SPLINE
SPL {X  -146.599, Y  +744.345, Z    +0.000, E1   -36.661, E3 +275980.416}
SPL {X  -158.886, Y  +709.076, Z    +0.000, E1   -22.176, E3 +275984.288}
SPL {X  -161.886, Y  +690.913, Z    +0.000, E1   -12.672, E3 +275988.922}
SPL {X  -162.573, Y  +682.458, Z    +0.000, E1    -7.683, E3 +275988.423}
SPL {X  -162.817, Y  +674.426, Z    +0.000, E1    -2.573, E3 +275988.141}
SPL {X  -162.820, Y  +670.554, Z    +0.000, E1    +0.472, E3 +275987.766}
SPL {X  -162.820, Y  +667.789, Z    +0.000, E1    +3.144, E3 +275987.787}
SPL {X  -162.820, Y  +664.083, Z    +0.000, E1    +7.387, E3 +275987.679}
SPL {X  -162.820, Y  +659.344, Z    +0.000, E1   +13.535, E3 +275987.243}
SPL {X  -162.820, Y  +653.403, Z    +0.000, E1   +21.415, E3 +275987.657}
SPL {X  -162.820, Y  +642.162, Z    +0.000, E1   +35.510, E3 +275986.970}
SPL {X  -162.820, Y  +598.675, Z    +0.000, E1   +56.845, E3 +276004.282}
SPL {X  -162.820, Y  +543.175, Z    +0.000, E1   +54.504, E3 +276080.137}
SPL {X  -162.820, Y  +538.115, Z    +0.000, E1   +53.658, E3 +276093.188}
SPL {X  -162.820, Y  +527.429, Z    +0.000, E1   +53.760, E3 +276108.918}
SPL {X  -162.820, Y  +518.365, Z    +0.000, E1   +53.683, E3 +276123.176}
SPL {X  -162.820, Y  +510.654, Z    +0.000, E1   +53.658, E3 +276135.175}
SPL {X  -162.820, Y  +501.304, Z    +0.000, E1   +53.758, E3 +276148.863}
SPL {X  -162.820, Y  +493.008, Z    +0.000, E1   +53.586, E3 +276162.639}
SPL {X  -162.820, Y  +484.615, Z    +0.000, E1   +53.726, E3 +276174.569}
ENDSPLINE

SPLINE
SPL {X  -162.820, Y  +492.996, Z    +0.000, E1   +49.430, E3 +276187.115}
ENDSPLINE

SPLINE
SPL {X  -162.820, Y  +486.578, Z    +0.000, E1   +49.194, E3 +276199.918}
SPL {X  -162.820, Y  +476.731, Z    +0.000, E1   +50.039, E3 +276212.341}
SPL {X  -162.820, Y  +466.442, Z    +0.000, E1   +50.873, E3 +276225.009}
SPL {X  -162.820, Y  +455.624, Z    +0.000, E1   +51.698, E3 +276238.081}
SPL {X  -162.820, Y  +444.568, Z    +0.000, E1   +52.608, E3 +276250.393}
SPL {X  -162.820, Y  +432.435, Z    +0.000, E1   +53.605, E3 +276263.276}
SPL {X  -162.820, Y  +419.900, Z    +0.000, E1   +54.598, E3 +276275.951}
SPL {X  -162.820, Y  +411.092, Z    +0.000, E1   +54.552, E3 +276289.471}
SPL {X  -162.820, Y  +400.244, Z    +0.000, E1   +54.630, E3 +276304.938}
SPL {X  -162.820, Y  +389.249, Z    +0.000, E1   +54.752, E3 +276320.517}
SPL {X  -162.820, Y  +380.650, Z    +0.000, E1   +54.601, E3 +276333.961}
SPL {X  -162.727, Y  +374.992, Z    +0.000, E1   +54.549, E3 +276342.644}
SPL {X  -162.216, Y  +366.490, Z    +0.000, E1   +54.549, E3 +276355.443}
SPL {X  -161.062, Y  +356.641, Z    +0.000, E1   +54.440, E3 +276370.561}
SPL {X  -159.761, Y  +349.086, Z    +0.000, E1   +54.132, E3 +276383.582}
SPL {X  -158.033, Y  +341.310, Z    +0.000, E1   +53.819, E3 +276396.972}
SPL {X  -156.195, Y  +334.528, Z    +0.000, E1   +53.534, E3 +276408.538}
SPL {X  -154.120, Y  +327.988, Z    +0.000, E1   +53.171, E3 +276420.395}
SPL {X  -151.310, Y  +320.369, Z    +0.000, E1   +52.706, E3 +276434.109}
SPL {X  -148.923, Y  +314.679, Z    +0.000, E1   +52.172, E3 +276445.194}
SPL {X  -146.846, Y  +310.168, Z    +0.000, E1   +51.697, E3 +276454.255}
SPL {X  -140.627, Y  +298.437, Z    +0.000, E1   +54.251, E3 +276458.514}
SPL {X  -122.064, Y  +272.747, Z    +0.000, E1   +48.156, E3 +276564.039}
ENDSPLINE

SPLINE
SPL {X  -148.173, Y  +313.009, Z    +0.000, E1   +35.624, E3 +276647.085}
SPL {X  -158.289, Y  +342.356, Z    +0.000, E1   +23.452, E3 +276650.074}
SPL {X  -161.301, Y  +358.312, Z    +0.000, E1   +15.384, E3 +276652.032}
SPL {X  -162.692, Y  +374.052, Z    +0.000, E1    +6.208, E3 +276651.970}
SPL {X  -162.820, Y  +381.030, Z    +0.000, E1    +1.454, E3 +276652.149}
SPL {X  -162.820, Y  +384.274, Z    +0.000, E1    -1.205, E3 +276651.868}
SPL {X  -162.820, Y  +388.271, Z    +0.000, E1    -5.458, E3 +276651.861}
SPL {X  -162.820, Y  +394.827, Z    +0.000, E1   -13.677, E3 +276651.551}
SPL {X  -162.820, Y  +402.977, Z    +0.000, E1   -24.772, E3 +276651.833}
SPL {X  -162.820, Y  +413.615, Z    +0.000, E1   -37.560, E3 +276651.623}
SPL {X  -162.820, Y  +456.390, Z    +0.000, E1   -57.415, E3 +276668.665}
SPL {X  -162.820, Y  +525.017, Z    +0.000, E1   -58.379, E3 +276739.329}
ENDSPLINE

SPLINE
SPL {X  -162.820, Y  +515.796, Z    +0.000, E1   -54.952, E3 +276748.436}
ENDSPLINE

SPLINE
SPL {X  -162.820, Y  +522.537, Z    +0.000, E1   -55.218, E3 +276756.611}
SPL {X  -162.820, Y  +529.742, Z    +0.000, E1   -55.146, E3 +276767.538}
SPL {X  -162.820, Y  +538.383, Z    +0.000, E1   -55.306, E3 +276778.990}
SPL {X  -162.820, Y  +544.790, Z    +0.000, E1   -55.066, E3 +276789.790}
SPL {X  -162.820, Y  +552.981, Z    +0.000, E1   -55.286, E3 +276800.253}
SPL {X  -162.820, Y  +560.767, Z    +0.000, E1   -55.137, E3 +276812.561}
SPL {X  -162.820, Y  +570.590, Z    +0.000, E1   -55.270, E3 +276825.895}
SPL {X  -162.820, Y  +577.946, Z    +0.000, E1   -55.110, E3 +276837.533}
SPL {X  -162.820, Y  +583.981, Z    +0.000, E1   -55.057, E3 +276846.615}
SPL {X  -162.820, Y  +591.604, Z    +0.000, E1   -55.202, E3 +276856.789}
SPL {X  -162.820, Y  +600.465, Z    +0.000, E1   -55.218, E3 +276869.578}
SPL {X  -162.820, Y  +609.951, Z    +0.000, E1   -55.211, E3 +276883.325}
SPL {X  -162.820, Y  +617.278, Z    +0.000, E1   -55.256, E3 +276893.549}
SPL {X  -162.820, Y  +625.209, Z    +0.000, E1   -55.167, E3 +276905.741}
SPL {X  -162.820, Y  +634.693, Z    +0.000, E1   -55.198, E3 +276919.197}
SPL {X  -162.820, Y  +642.452, Z    +0.000, E1   -55.141, E3 +276930.804}
SPL {X  -162.820, Y  +652.837, Z    +0.000, E1   -55.281, E3 +276945.072}
SPL {X  -162.820, Y  +660.849, Z    +0.000, E1   -55.101, E3 +276957.621}
SPL {X  -162.820, Y  +668.534, Z    +0.000, E1   -55.182, E3 +276968.334}
SPL {X  -162.763, Y  +677.803, Z    +0.000, E1   -55.175, E3 +276981.840}
SPL {X  -162.314, Y  +686.325, Z    +0.000, E1   -55.173, E3 +276994.121}
SPL {X  -161.784, Y  +691.841, Z    +0.000, E1   -55.010, E3 +277003.083}
SPL {X  -161.070, Y  +697.305, Z    +0.000, E1   -54.828, E3 +277012.161}
SPL {X  -159.751, Y  +704.965, Z    +0.000, E1   -54.697, E3 +277024.147}
SPL {X  -158.271, Y  +711.718, Z    +0.000, E1   -54.504, E3 +277034.955}
SPL {X  -157.115, Y  +716.223, Z    +0.000, E1   -54.227, E3 +277043.147}
SPL {X  -154.825, Y  +723.894, Z    +0.000, E1   -53.830, E3 +277056.687}
SPL {X  -152.160, Y  +731.445, Z    +0.000, E1   -53.336, E3 +277070.229}
SPL {X  -149.361, Y  +738.321, Z    +0.000, E1   -52.873, E3 +277082.692}
SPL {X  -146.885, Y  +743.751, Z    +0.000, E1   -52.544, E3 +277092.053}
SPL {X  -144.373, Y  +748.778, Z    +0.000, E1   -52.887, E3 +277097.515}
SPL {X  -137.947, Y  +759.993, Z    +0.000, E1   -55.381, E3 +277100.625}
SPL {X  -123.111, Y  +780.056, Z    +0.000, E1   -48.144, E3 +277199.761}
ENDSPLINE

SPLINE
SPL {X  -146.599, Y  +744.345, Z    +0.000, E1   -36.661, E3 +277284.764}
SPL {X  -157.185, Y  +715.965, Z    +0.000, E1   -25.340, E3 +277287.814}
SPL {X  -159.997, Y  +703.690, Z    +0.000, E1   -19.457, E3 +277289.142}
SPL {X  -161.886, Y  +690.913, Z    +0.000, E1   -12.672, E3 +277293.270}
SPL {X  -162.700, Y  +679.756, Z    +0.000, E1    -6.060, E3 +277292.479}
SPL {X  -162.820, Y  +673.439, Z    +0.000, E1    -1.797, E3 +277292.581}
SPL {X  -162.820, Y  +670.554, Z    +0.000, E1    +0.472, E3 +277292.114}
SPL {X  -162.820, Y  +667.789, Z    +0.000, E1    +3.144, E3 +277292.135}
SPL {X  -162.820, Y  +664.083, Z    +0.000, E1    +7.387, E3 +277292.027}
SPL {X  -162.820, Y  +659.344, Z    +0.000, E1   +13.535, E3 +277291.591}
SPL {X  -162.820, Y  +653.403, Z    +0.000, E1   +21.415, E3 +277292.005}
SPL {X  -162.820, Y  +642.162, Z    +0.000, E1   +35.510, E3 +277291.318}
SPL {X  -162.820, Y  +598.675, Z    +0.000, E1   +56.845, E3 +277308.630}
SPL {X  -162.820, Y  +543.175, Z    +0.000, E1   +54.504, E3 +277384.485}
SPL {X  -162.820, Y  +538.115, Z    +0.000, E1   +53.658, E3 +277397.536}
SPL {X  -162.820, Y  +530.332, Z    +0.000, E1   +53.757, E3 +277408.679}
SPL {X  -162.820, Y  +525.300, Z    +0.000, E1   +53.701, E3 +277416.730}
SPL {X  -162.820, Y  +518.365, Z    +0.000, E1   +53.683, E3 +277427.524}
SPL {X  -162.820, Y  +510.654, Z    +0.000, E1   +53.658, E3 +277439.523}
SPL {X  -162.820, Y  +501.304, Z    +0.000, E1   +53.758, E3 +277453.211}
SPL {X  -162.820, Y  +493.008, Z    +0.000, E1   +53.586, E3 +277466.986}
SPL {X  -162.820, Y  +484.615, Z    +0.000, E1   +53.726, E3 +277478.917}
ENDSPLINE

SPLINE
SPL {X  -162.820, Y  +492.996, Z    +0.000, E1   +49.430, E3 +277491.463}
ENDSPLINE

SPLINE
SPL {X  -162.820, Y  +486.578, Z    +0.000, E1   +49.194, E3 +277504.266}
SPL {X  -162.820, Y  +476.731, Z    +0.000, E1   +50.039, E3 +277516.689}
SPL {X  -162.820, Y  +466.442, Z    +0.000, E1   +50.873, E3 +277529.357}
SPL {X  -162.820, Y  +455.624, Z    +0.000, E1   +51.698, E3 +277542.428}
SPL {X  -162.820, Y  +444.568, Z    +0.000, E1   +52.608, E3 +277554.741}
SPL {X  -162.820, Y  +432.435, Z    +0.000, E1   +53.605, E3 +277567.624}
SPL {X  -162.820, Y  +419.875, Z    +0.000, E1   +54.604, E3 +277580.298}
SPL {X  -162.820, Y  +414.181, Z    +0.000, E1   +54.446, E3 +277589.733}
SPL {X  -162.820, Y  +407.616, Z    +0.000, E1   +54.585, E3 +277598.567}
SPL {X  -162.820, Y  +400.244, Z    +0.000, E1   +54.630, E3 +277609.285}
SPL {X  -162.820, Y  +389.249, Z    +0.000, E1   +54.752, E3 +277624.864}
SPL {X  -162.820, Y  +380.650, Z    +0.000, E1   +54.601, E3 +277638.309}
SPL {X  -162.727, Y  +374.992, Z    +0.000, E1   +54.549, E3 +277646.991}
SPL {X  -162.373, Y  +368.447, Z    +0.000, E1   +54.597, E3 +277656.424}
SPL {X  -161.939, Y  +363.587, Z    +0.000, E1   +54.355, E3 +277665.036}
SPL {X  -160.880, Y  +355.442, Z    +0.000, E1   +54.372, E3 +277677.247}
SPL {X  -159.457, Y  +347.579, Z    +0.000, E1   +54.148, E3 +277689.983}
SPL {X  -158.033, Y  +341.310, Z    +0.000, E1   +53.819, E3 +277701.320}
SPL {X  -156.195, Y  +334.528, Z    +0.000, E1   +53.534, E3 +277712.885}
SPL {X  -154.120, Y  +327.988, Z    +0.000, E1   +53.171, E3 +277724.742}
SPL {X  -151.310, Y  +320.369, Z    +0.000, E1   +52.706, E3 +277738.457}
SPL {X  -148.923, Y  +314.679, Z    +0.000, E1   +52.172, E3 +277749.542}
SPL {X  -146.846, Y  +310.168, Z    +0.000, E1   +51.697, E3 +277758.603}
SPL {X  -140.627, Y  +298.437, Z    +0.000, E1   +54.251, E3 +277762.862}
SPL {X  -122.064, Y  +272.747, Z    +0.000, E1   +48.156, E3 +277868.387}
ENDSPLINE

SPLINE
SPL {X  -148.173, Y  +313.009, Z    +0.000, E1   +35.624, E3 +277951.433}
SPL {X  -159.343, Y  +347.032, Z    +0.000, E1   +21.245, E3 +277955.276}
SPL {X  -161.787, Y  +362.186, Z    +0.000, E1   +13.182, E3 +277956.472}
SPL {X  -162.692, Y  +374.052, Z    +0.000, E1    +6.208, E3 +277956.318}
SPL {X  -162.820, Y  +381.030, Z    +0.000, E1    +1.454, E3 +277956.497}
SPL {X  -162.820, Y  +384.274, Z    +0.000, E1    -1.205, E3 +277956.216}
SPL {X  -162.820, Y  +388.271, Z    +0.000, E1    -5.458, E3 +277956.209}
SPL {X  -162.820, Y  +394.827, Z    +0.000, E1   -13.677, E3 +277955.899}
SPL {X  -162.820, Y  +402.977, Z    +0.000, E1   -24.772, E3 +277956.180}
SPL {X  -162.820, Y  +413.615, Z    +0.000, E1   -37.560, E3 +277955.971}
SPL {X  -162.820, Y  +452.521, Z    +0.000, E1   -56.942, E3 +277970.263}
SPL {X  -162.820, Y  +459.967, Z    +0.000, E1   -57.801, E3 +277975.559}
SPL {X  -162.820, Y  +525.017, Z    +0.000, E1   -58.379, E3 +278043.677}
ENDSPLINE

SPLINE
SPL {X  -162.820, Y  +515.796, Z    +0.000, E1   -54.952, E3 +278052.784}
ENDSPLINE

SPLINE
SPL {X  -162.820, Y  +522.537, Z    +0.000, E1   -55.218, E3 +278060.959}
SPL {X  -162.820, Y  +529.742, Z    +0.000, E1   -55.146, E3 +278071.886}
SPL {X  -162.820, Y  +538.383, Z    +0.000, E1   -55.306, E3 +278083.338}
SPL {X  -162.820, Y  +544.790, Z    +0.000, E1   -55.066, E3 +278094.138}
SPL {X  -162.820, Y  +552.981, Z    +0.000, E1   -55.286, E3 +278104.601}
SPL {X  -162.820, Y  +560.767, Z    +0.000, E1   -55.137, E3 +278116.909}
SPL {X  -162.820, Y  +570.590, Z    +0.000, E1   -55.270, E3 +278130.243}
SPL {X  -162.820, Y  +580.865, Z    +0.000, E1   -55.132, E3 +278146.200}
SPL {X  -162.820, Y  +591.604, Z    +0.000, E1   -55.202, E3 +278161.137}
SPL {X  -162.820, Y  +600.465, Z    +0.000, E1   -55.218, E3 +278173.926}
SPL {X  -162.820, Y  +609.951, Z    +0.000, E1   -55.211, E3 +278187.673}
SPL {X  -162.820, Y  +618.960, Z    +0.000, E1   -55.186, E3 +278200.893}
SPL {X  -162.820, Y  +627.322, Z    +0.000, E1   -55.201, E3 +278212.829}
SPL {X  -162.820, Y  +634.693, Z    +0.000, E1   -55.198, E3 +278223.545}
SPL {X  -162.820, Y  +642.452, Z    +0.000, E1   -55.141, E3 +278235.152}
SPL {X  -162.820, Y  +649.370, Z    +0.000, E1   -55.160, E3 +278245.009}
SPL {X  -162.820, Y  +658.542, Z    +0.000, E1   -55.251, E3 +278257.887}
SPL {X  -162.820, Y  +668.534, Z    +0.000, E1   -55.182, E3 +278272.682}
SPL {X  -162.763, Y  +677.803, Z    +0.000, E1   -55.175, E3 +278286.188}
SPL {X  -162.314, Y  +686.325, Z    +0.000, E1   -55.173, E3 +278298.469}
SPL {X  -161.784, Y  +691.841, Z    +0.000, E1   -55.010, E3 +278307.431}
SPL {X  -161.070, Y  +697.305, Z    +0.000, E1   -54.828, E3 +278316.509}
SPL {X  -159.751, Y  +704.965, Z    +0.000, E1   -54.697, E3 +278328.495}
SPL {X  -158.271, Y  +711.718, Z    +0.000, E1   -54.504, E3 +278339.303}
SPL {X  -157.115, Y  +716.223, Z    +0.000, E1   -54.227, E3 +278347.495}
SPL {X  -155.622, Y  +721.376, Z    +0.000, E1   -53.849, E3 +278357.095}
SPL {X  -153.323, Y  +728.294, Z    +0.000, E1   -53.618, E3 +278368.568}
SPL {X  -150.606, Y  +735.372, Z    +0.000, E1   -53.091, E3 +278381.565}
SPL {X  -148.712, Y  +739.795, Z    +0.000, E1   -52.656, E3 +278390.127}
SPL {X  -146.885, Y  +743.751, Z    +0.000, E1   -52.544, E3 +278396.401}
SPL {X  -144.373, Y  +748.778, Z    +0.000, E1   -52.887, E3 +278401.863}
SPL {X  -137.947, Y  +759.993, Z    +0.000, E1   -55.381, E3 +278404.973}
SPL {X  -123.111, Y  +780.056, Z    +0.000, E1   -48.144, E3 +278504.109}
ENDSPLINE

SPLINE
SPL {X  -146.599, Y  +744.345, Z    +0.000, E1   -36.661, E3 +278589.112}
SPL {X  -158.886, Y  +709.076, Z    +0.000, E1   -22.176, E3 +278592.984}
SPL {X  -161.886, Y  +690.913, Z    +0.000, E1   -12.672, E3 +278597.618}
SPL {X  -162.573, Y  +682.458, Z    +0.000, E1    -7.683, E3 +278597.119}
SPL {X  -162.817, Y  +674.426, Z    +0.000, E1    -2.573, E3 +278596.837}
SPL {X  -162.820, Y  +670.554, Z    +0.000, E1    +0.472, E3 +278596.461}
SPL {X  -162.820, Y  +667.789, Z    +0.000, E1    +3.144, E3 +278596.483}
SPL {X  -162.820, Y  +664.083, Z    +0.000, E1    +7.387, E3 +278596.375}
SPL {X  -162.820, Y  +659.344, Z    +0.000, E1   +13.535, E3 +278595.939}
SPL {X  -162.820, Y  +653.403, Z    +0.000, E1   +21.415, E3 +278596.353}
SPL {X  -162.820, Y  +642.162, Z    +0.000, E1   +35.510, E3 +278595.666}
SPL {X  -162.820, Y  +598.675, Z    +0.000, E1   +56.845, E3 +278612.978}
SPL {X  -162.820, Y  +543.175, Z    +0.000, E1   +54.504, E3 +278688.833}
SPL {X  -162.820, Y  +538.115, Z    +0.000, E1   +53.658, E3 +278701.884}
SPL {X  -162.820, Y  +527.429, Z    +0.000, E1   +53.760, E3 +278717.614}
SPL {X  -162.820, Y  +518.365, Z    +0.000, E1   +53.683, E3 +278731.871}
SPL {X  -162.820, Y  +510.654, Z    +0.000, E1   +53.658, E3 +278743.870}
SPL {X  -162.820, Y  +501.304, Z    +0.000, E1   +53.758, E3 +278757.559}
SPL {X  -162.820, Y  +493.008, Z    +0.000, E1   +53.586, E3 +278771.334}
SPL {X  -162.820, Y  +484.615, Z    +0.000, E1   +53.726, E3 +278783.265}
ENDSPLINE

SPLINE
SPL {X  -162.820, Y  +492.996, Z    +0.000, E1   +49.430, E3 +278795.811}
ENDSPLINE

SPLINE
SPL {X  -162.820, Y  +483.544, Z    +0.000, E1   +49.458, E3 +278812.596}
SPL {X  -162.820, Y  +468.441, Z    +0.000, E1   +50.759, E3 +278831.098}
SPL {X  -162.820, Y  +455.624, Z    +0.000, E1   +51.698, E3 +278846.776}
SPL {X  -162.820, Y  +444.568, Z    +0.000, E1   +52.608, E3 +278859.089}
SPL {X  -162.820, Y  +432.435, Z    +0.000, E1   +53.605, E3 +278871.972}
SPL {X  -162.820, Y  +419.875, Z    +0.000, E1   +54.604, E3 +278884.646}
SPL {X  -162.820, Y  +414.181, Z    +0.000, E1   +54.446, E3 +278894.081}
SPL {X  -162.820, Y  +407.616, Z    +0.000, E1   +54.585, E3 +278902.915}
SPL {X  -162.820, Y  +400.244, Z    +0.000, E1   +54.630, E3 +278913.633}
SPL {X  -162.820, Y  +389.249, Z    +0.000, E1   +54.752, E3 +278929.212}
SPL {X  -162.799, Y  +377.862, Z    +0.000, E1   +54.622, E3 +278946.843}
SPL {X  -162.216, Y  +366.490, Z    +0.000, E1   +54.549, E3 +278964.138}
SPL {X  -160.880, Y  +355.442, Z    +0.000, E1   +54.372, E3 +278981.595}
SPL {X  -159.457, Y  +347.579, Z    +0.000, E1   +54.148, E3 +278994.331}
SPL {X  -158.033, Y  +341.310, Z    +0.000, E1   +53.819, E3 +279005.668}
SPL {X  -155.608, Y  +332.578, Z    +0.000, E1   +53.425, E3 +279020.939}
SPL {X  -152.785, Y  +324.223, Z    +0.000, E1   +52.975, E3 +279035.699}
SPL {X  -150.663, Y  +318.766, Z    +0.000, E1   +52.574, E3 +279045.732}
SPL {X  -148.923, Y  +314.679, Z    +0.000, E1   +52.172, E3 +279053.890}
SPL {X  -146.846, Y  +310.168, Z    +0.000, E1   +51.697, E3 +279062.951}
SPL {X  -140.627, Y  +298.437, Z    +0.000, E1   +54.251, E3 +279067.210}
SPL {X  -122.064, Y  +272.747, Z    +0.000, E1   +48.156, E3 +279172.735}
ENDSPLINE

SPLINE
SPL {X  -148.173, Y  +313.009, Z    +0.000, E1   +35.624, E3 +279255.781}
SPL {X  -158.289, Y  +342.356, Z    +0.000, E1   +23.452, E3 +279258.770}
SPL {X  -161.301, Y  +358.312, Z    +0.000, E1   +15.384, E3 +279260.728}
SPL {X  -162.692, Y  +374.052, Z    +0.000, E1    +6.208, E3 +279260.666}
SPL {X  -162.820, Y  +381.030, Z    +0.000, E1    +1.454, E3 +279260.845}
SPL {X  -162.820, Y  +383.414, Z    +0.000, E1    -0.499, E3 +279260.751}
SPL {X  -162.820, Y  +385.887, Z    +0.000, E1    -2.819, E3 +279260.473}
SPL {X  -162.820, Y  +389.383, Z    +0.000, E1    -6.871, E3 +279260.540}
SPL {X  -162.820, Y  +393.153, Z    +0.000, E1   -11.600, E3 +279260.433}
SPL {X  -162.820, Y  +400.748, Z    +0.000, E1   -21.791, E3 +279260.225}
SPL {X  -162.820, Y  +413.615, Z    +0.000, E1   -37.560, E3 +279260.319}
SPL {X  -162.820, Y  +456.390, Z    +0.000, E1   -57.415, E3 +279277.360}
SPL {X  -162.820, Y  +525.017, Z    +0.000, E1   -58.379, E3 +279348.025}
ENDSPLINE

SPLINE
SPL {X  -162.820, Y  +520.266, Z    +0.000, E1   -55.155, E3 +279362.518}
ENDSPLINE

SPLINE
SPL {X  -162.820, Y  +529.742, Z    +0.000, E1   -55.146, E3 +279376.234}
SPL {X  -162.820, Y  +538.383, Z    +0.000, E1   -55.306, E3 +279387.686}
SPL {X  -162.820, Y  +544.790, Z    +0.000, E1   -55.066, E3 +279398.486}
SPL {X  -162.820, Y  +552.981, Z    +0.000, E1   -55.286, E3 +279408.949}
SPL {X  -162.820, Y  +560.767, Z    +0.000, E1   -55.137, E3 +279421.257}
SPL {X  -162.820, Y  +570.590, Z    +0.000, E1   -55.270, E3 +279434.591}
SPL {X  -162.820, Y  +577.946, Z    +0.000, E1   -55.110, E3 +279446.229}
SPL {X  -162.820, Y  +583.981, Z    +0.000, E1   -55.057, E3 +279455.311}
SPL {X  -162.820, Y  +594.246, Z    +0.000, E1   -55.310, E3 +279468.747}
SPL {X  -162.820, Y  +601.811, Z    +0.000, E1   -55.027, E3 +279481.274}
SPL {X  -162.820, Y  +609.951, Z    +0.000, E1   -55.211, E3 +279492.021}
SPL {X  -162.820, Y  +618.960, Z    +0.000, E1   -55.186, E3 +279505.241}
SPL {X  -162.820, Y  +627.322, Z    +0.000, E1   -55.201, E3 +279517.176}
SPL {X  -162.820, Y  +634.693, Z    +0.000, E1   -55.198, E3 +279527.893}
SPL {X  -162.820, Y  +642.452, Z    +0.000, E1   -55.141, E3 +279539.500}
SPL {X  -162.820, Y  +652.837, Z    +0.000, E1   -55.281, E3 +279553.768}
SPL {X  -162.820, Y  +660.849, Z    +0.000, E1   -55.101, E3 +279566.317}
SPL {X  -162.820, Y  +668.534, Z    +0.000, E1   -55.182, E3 +279577.030}
SPL {X  -162.763, Y  +677.803, Z    +0.000, E1   -55.175, E3 +279590.536}
SPL {X  -162.314, Y  +686.325, Z    +0.000, E1   -55.173, E3 +279602.816}
SPL {X  -161.784, Y  +691.841, Z    +0.000, E1   -55.010, E3 +279611.778}
SPL {X  -161.070, Y  +697.305, Z    +0.000, E1   -54.828, E3 +279620.856}
SPL {X  -159.751, Y  +704.965, Z    +0.000, E1   -54.697, E3 +279632.842}
SPL {X  -158.271, Y  +711.718, Z    +0.000, E1   -54.504, E3 +279643.651}
SPL {X  -157.115, Y  +716.223, Z    +0.000, E1   -54.227, E3 +279651.843}
SPL {X  -155.622, Y  +721.376, Z    +0.000, E1   -53.849, E3 +279661.443}
SPL {X  -153.323, Y  +728.294, Z    +0.000, E1   -53.618, E3 +279672.916}
SPL {X  -150.606, Y  +735.372, Z    +0.000, E1   -53.091, E3 +279685.912}
SPL {X  -148.712, Y  +739.795, Z    +0.000, E1   -52.656, E3 +279694.475}
SPL {X  -146.885, Y  +743.751, Z    +0.000, E1   -52.544, E3 +279700.748}
SPL {X  -144.373, Y  +748.778, Z    +0.000, E1   -52.887, E3 +279706.211}
SPL {X  -137.947, Y  +759.993, Z    +0.000, E1   -55.381, E3 +279709.321}
SPL {X  -123.111, Y  +780.056, Z    +0.000, E1   -48.144, E3 +279808.456}
ENDSPLINE

SPLINE
SPL {X  -146.599, Y  +744.345, Z    +0.000, E1   -36.661, E3 +279893.460}
SPL {X  -158.886, Y  +709.076, Z    +0.000, E1   -22.176, E3 +279897.332}
SPL {X  -161.886, Y  +690.913, Z    +0.000, E1   -12.672, E3 +279901.966}
SPL {X  -162.573, Y  +682.458, Z    +0.000, E1    -7.683, E3 +279901.467}
SPL {X  -162.817, Y  +674.426, Z    +0.000, E1    -2.573, E3 +279901.185}
SPL {X  -162.820, Y  +670.554, Z    +0.000, E1    +0.472, E3 +279900.809}
SPL {X  -162.820, Y  +667.789, Z    +0.000, E1    +3.144, E3 +279900.831}
SPL {X  -162.820, Y  +664.083, Z    +0.000, E1    +7.387, E3 +279900.723}
SPL {X  -162.820, Y  +659.344, Z    +0.000, E1   +13.535, E3 +279900.286}
SPL {X  -162.820, Y  +653.403, Z    +0.000, E1   +21.415, E3 +279900.701}
SPL {X  -162.820, Y  +644.970, Z    +0.000, E1   +32.346, E3 +279900.117}
SPL {X  -162.820, Y  +637.013, Z    +0.000, E1   +41.185, E3 +279899.822}
SPL {X  -162.820, Y  +603.840, Z    +0.000, E1   +55.833, E3 +279914.439}
SPL {X  -162.820, Y  +590.612, Z    +0.000, E1   +58.217, E3 +279921.823}
SPL {X  -162.820, Y  +543.175, Z    +0.000, E1   +54.504, E3 +279993.180}
SPL {X  -162.820, Y  +538.115, Z    +0.000, E1   +53.658, E3 +280006.232}
SPL {X  -162.820, Y  +527.429, Z    +0.000, E1   +53.760, E3 +280021.961}
SPL {X  -162.820, Y  +518.365, Z    +0.000, E1   +53.683, E3 +280036.219}
SPL {X  -162.820, Y  +510.654, Z    +0.000, E1   +53.658, E3 +280048.218}
SPL {X  -162.820, Y  +501.304, Z    +0.000, E1   +53.758, E3 +280061.907}
SPL {X  -162.820, Y  +493.008, Z    +0.000, E1   +53.586, E3 +280075.682}
SPL {X  -162.820, Y  +485.759, Z    +0.000, E1   +53.138, E3 +280089.690}
ENDSPLINE

SPLINE
SPL {X  -162.820, Y  +494.645, Z    +0.000, E1   +48.544, E3 +280102.165}
ENDSPLINE

SPLINE
SPL {X  -162.820, Y  +486.578, Z    +0.000, E1   +49.194, E3 +280112.962}
SPL {X  -162.820, Y  +476.731, Z    +0.000, E1   +50.039, E3 +280125.384}
SPL {X  -162.820, Y  +466.442, Z    +0.000, E1   +50.873, E3 +280138.053}
SPL {X  -162.820, Y  +455.624, Z    +0.000, E1   +51.698, E3 +280151.124}
SPL {X  -162.820, Y  +444.568, Z    +0.000, E1   +52.608, E3 +280163.437}
SPL {X  -162.820, Y  +432.435, Z    +0.000, E1   +53.605, E3 +280176.320}
SPL {X  -162.820, Y  +419.900, Z    +0.000, E1   +54.598, E3 +280188.995}
SPL {X  -162.820, Y  +411.092, Z    +0.000, E1   +54.552, E3 +280202.514}
SPL {X  -162.820, Y  +400.244, Z    +0.000, E1   +54.630, E3 +280217.981}
SPL {X  -162.820, Y  +392.496, Z    +0.000, E1   +54.734, E3 +280228.682}
SPL {X  -162.820, Y  +387.085, Z    +0.000, E1   +54.699, E3 +280236.909}
SPL {X  -162.820, Y  +380.650, Z    +0.000, E1   +54.601, E3 +280247.005}
SPL {X  -162.727, Y  +374.992, Z    +0.000, E1   +54.549, E3 +280255.687}
SPL {X  -162.216, Y  +366.490, Z    +0.000, E1   +54.549, E3 +280268.486}
SPL {X  -160.880, Y  +355.442, Z    +0.000, E1   +54.372, E3 +280285.942}
SPL {X  -159.457, Y  +347.579, Z    +0.000, E1   +54.148, E3 +280298.679}
SPL {X  -158.033, Y  +341.310, Z    +0.000, E1   +53.819, E3 +280310.015}
SPL {X  -155.608, Y  +332.578, Z    +0.000, E1   +53.425, E3 +280325.287}
SPL {X  -153.385, Y  +325.878, Z    +0.000, E1   +53.068, E3 +280336.955}
SPL {X  -151.310, Y  +320.369, Z    +0.000, E1   +52.706, E3 +280347.153}
SPL {X  -148.923, Y  +314.679, Z    +0.000, E1   +52.172, E3 +280358.237}
SPL {X  -146.846, Y  +310.168, Z    +0.000, E1   +51.697, E3 +280367.299}
SPL {X  -140.627, Y  +298.437, Z    +0.000, E1   +54.251, E3 +280371.557}
SPL {X  -122.064, Y  +272.747, Z    +0.000, E1   +48.156, E3 +280477.083}
ENDSPLINE

SPLINE
SPL {X  -148.173, Y  +313.009, Z    +0.000, E1   +35.624, E3 +280560.128}
SPL {X  -158.289, Y  +342.356, Z    +0.000, E1   +23.452, E3 +280563.118}
SPL {X  -161.301, Y  +358.312, Z    +0.000, E1   +15.384, E3 +280565.075}
SPL {X  -162.692, Y  +374.052, Z    +0.000, E1    +6.208, E3 +280565.014}
SPL {X  -162.820, Y  +381.030, Z    +0.000, E1    +1.454, E3 +280565.193}
SPL {X  -162.820, Y  +384.274, Z    +0.000, E1    -1.205, E3 +280564.912}
SPL {X  -162.820, Y  +388.271, Z    +0.000, E1    -5.458, E3 +280564.904}
SPL {X  -162.820, Y  +394.827, Z    +0.000, E1   -13.677, E3 +280564.594}
SPL {X  -162.820, Y  +402.977, Z    +0.000, E1   -24.772, E3 +280564.876}
SPL {X  -162.820, Y  +413.615, Z    +0.000, E1   -37.560, E3 +280564.667}
SPL {X  -162.820, Y  +456.390, Z    +0.000, E1   -57.415, E3 +280581.708}
SPL {X  -162.820, Y  +525.017, Z    +0.000, E1   -58.379, E3 +280652.373}
ENDSPLINE

SPLINE
SPL {X  -162.820, Y  +515.796, Z    +0.000, E1   -54.952, E3 +280661.479}
ENDSPLINE

SPLINE
SPL {X  -162.820, Y  +522.537, Z    +0.000, E1   -55.218, E3 +280669.654}
SPL {X  -162.820, Y  +529.742, Z    +0.000, E1   -55.146, E3 +280680.582}
SPL {X  -162.820, Y  +538.383, Z    +0.000, E1   -55.306, E3 +280692.034}
SPL {X  -162.820, Y  +544.790, Z    +0.000, E1   -55.066, E3 +280702.834}
SPL {X  -162.820, Y  +552.981, Z    +0.000, E1   -55.286, E3 +280713.296}
SPL {X  -162.820, Y  +560.767, Z    +0.000, E1   -55.137, E3 +280725.605}
SPL {X  -162.820, Y  +570.590, Z    +0.000, E1   -55.270, E3 +280738.939}
SPL {X  -162.820, Y  +577.946, Z    +0.000, E1   -55.110, E3 +280750.577}
SPL {X  -162.820, Y  +583.981, Z    +0.000, E1   -55.057, E3 +280759.659}
SPL {X  -162.820, Y  +591.604, Z    +0.000, E1   -55.202, E3 +280769.833}
SPL {X  -162.820, Y  +600.465, Z    +0.000, E1   -55.218, E3 +280782.621}
SPL {X  -162.820, Y  +609.951, Z    +0.000, E1   -55.211, E3 +280796.369}
SPL {X  -162.820, Y  +617.278, Z    +0.000, E1   -55.256, E3 +280806.593}
SPL {X  -162.820, Y  +625.209, Z    +0.000, E1   -55.167, E3 +280818.785}
SPL {X  -162.820, Y  +634.693, Z    +0.000, E1   -55.198, E3 +280832.241}
SPL {X  -162.820, Y  +642.452, Z    +0.000, E1   -55.141, E3 +280843.847}
SPL {X  -162.820, Y  +652.837, Z    +0.000, E1   -55.281, E3 +280858.115}
SPL {X  -162.820, Y  +660.849, Z    +0.000, E1   -55.101, E3 +280870.664}
SPL {X  -162.820, Y  +668.534, Z    +0.000, E1   -55.182, E3 +280881.378}
SPL {X  -162.763, Y  +677.803, Z    +0.000, E1   -55.175, E3 +280894.884}
SPL {X  -162.314, Y  +686.325, Z    +0.000, E1   -55.173, E3 +280907.164}
SPL {X  -161.784, Y  +691.841, Z    +0.000, E1   -55.010, E3 +280916.126}
SPL {X  -161.070, Y  +697.305, Z    +0.000, E1   -54.828, E3 +280925.204}
SPL {X  -159.751, Y  +704.965, Z    +0.000, E1   -54.697, E3 +280937.190}
SPL {X  -158.271, Y  +711.718, Z    +0.000, E1   -54.504, E3 +280947.999}
SPL {X  -157.115, Y  +716.223, Z    +0.000, E1   -54.227, E3 +280956.190}
SPL {X  -154.825, Y  +723.894, Z    +0.000, E1   -53.830, E3 +280969.731}
SPL {X  -152.160, Y  +731.445, Z    +0.000, E1   -53.336, E3 +280983.273}
SPL {X  -149.361, Y  +738.321, Z    +0.000, E1   -52.873, E3 +280995.735}
SPL {X  -146.885, Y  +743.751, Z    +0.000, E1   -52.544, E3 +281005.096}
SPL {X  -144.373, Y  +748.778, Z    +0.000, E1   -52.887, E3 +281010.559}
SPL {X  -137.947, Y  +759.993, Z    +0.000, E1   -55.381, E3 +281013.668}
SPL {X  -123.111, Y  +780.056, Z    +0.000, E1   -48.144, E3 +281112.804}
ENDSPLINE

SPLINE
SPL {X  -146.599, Y  +744.345, Z    +0.000, E1   -36.661, E3 +281197.807}
SPL {X  -157.185, Y  +715.965, Z    +0.000, E1   -25.340, E3 +281200.857}
SPL {X  -159.997, Y  +703.690, Z    +0.000, E1   -19.457, E3 +281202.186}
SPL {X  -161.886, Y  +690.913, Z    +0.000, E1   -12.672, E3 +281206.314}
SPL {X  -162.700, Y  +679.756, Z    +0.000, E1    -6.060, E3 +281205.523}
SPL {X  -162.820, Y  +673.439, Z    +0.000, E1    -1.797, E3 +281205.625}
SPL {X  -162.820, Y  +670.554, Z    +0.000, E1    +0.472, E3 +281205.157}
SPL {X  -162.820, Y  +667.789, Z    +0.000, E1    +3.144, E3 +281205.179}
SPL {X  -162.820, Y  +664.083, Z    +0.000, E1    +7.387, E3 +281205.070}
SPL {X  -162.820, Y  +659.344, Z    +0.000, E1   +13.535, E3 +281204.634}
SPL {X  -162.820, Y  +653.403, Z    +0.000, E1   +21.415, E3 +281205.049}
SPL {X  -162.820, Y  +642.162, Z    +0.000, E1   +35.510, E3 +281204.361}
SPL {X  -162.820, Y  +598.675, Z    +0.000, E1   +56.845, E3 +281221.674}
SPL {X  -162.820, Y  +543.175, Z    +0.000, E1   +54.504, E3 +281297.528}
SPL {X  -162.820, Y  +538.115, Z    +0.000, E1   +53.658, E3 +281310.580}
SPL {X  -162.820, Y  +530.332, Z    +0.000, E1   +53.757, E3 +281321.723}
SPL {X  -162.820, Y  +525.300, Z    +0.000, E1   +53.701, E3 +281329.773}
SPL {X  -162.820, Y  +518.365, Z    +0.000, E1   +53.683, E3 +281340.567}
SPL {X  -162.820, Y  +510.654, Z    +0.000, E1   +53.658, E3 +281352.566}
SPL {X  -162.820, Y  +501.304, Z    +0.000, E1   +53.758, E3 +281366.255}
SPL {X  -162.820, Y  +493.008, Z    +0.000, E1   +53.586, E3 +281380.030}
SPL {X  -162.820, Y  +484.615, Z    +0.000, E1   +53.726, E3 +281391.961}
ENDSPLINE

SPLINE
SPL {X  -162.820, Y  +492.996, Z    +0.000, E1   +49.430, E3 +281404.507}
ENDSPLINE

SPLINE
SPL {X  -162.820, Y  +486.578, Z    +0.000, E1   +49.194, E3 +281417.309}
SPL {X  -162.820, Y  +476.731, Z    +0.000, E1   +50.039, E3 +281429.732}
SPL {X  -162.820, Y  +466.442, Z    +0.000, E1   +50.873, E3 +281442.401}
SPL {X  -162.820, Y  +455.624, Z    +0.000, E1   +51.698, E3 +281455.472}
SPL {X  -162.820, Y  +444.568, Z    +0.000, E1   +52.608, E3 +281467.785}
SPL {X  -162.820, Y  +432.435, Z    +0.000, E1   +53.605, E3 +281480.668}
SPL {X  -162.820, Y  +419.875, Z    +0.000, E1   +54.604, E3 +281493.342}
SPL {X  -162.820, Y  +414.181, Z    +0.000, E1   +54.446, E3 +281502.776}
SPL {X  -162.820, Y  +407.616, Z    +0.000, E1   +54.585, E3 +281511.611}
SPL {X  -162.820, Y  +400.244, Z    +0.000, E1   +54.630, E3 +281522.329}
SPL {X  -162.820, Y  +389.249, Z    +0.000, E1   +54.752, E3 +281537.908}
SPL {X  -162.820, Y  +380.650, Z    +0.000, E1   +54.601, E3 +281551.353}
SPL {X  -162.727, Y  +374.992, Z    +0.000, E1   +54.549, E3 +281560.035}
SPL {X  -162.373, Y  +368.447, Z    +0.000, E1   +54.597, E3 +281569.467}
SPL {X  -161.939, Y  +363.587, Z    +0.000, E1   +54.355, E3 +281578.079}
SPL {X  -161.062, Y  +356.641, Z    +0.000, E1   +54.440, E3 +281587.952}
SPL {X  -159.761, Y  +349.086, Z    +0.000, E1   +54.132, E3 +281600.973}
SPL {X  -158.451, Y  +343.033, Z    +0.000, E1   +53.828, E3 +281611.650}
SPL {X  -156.619, Y  +335.993, Z    +0.000, E1   +53.639, E3 +281623.296}
SPL {X  -154.959, Y  +330.520, Z    +0.000, E1   +53.198, E3 +281633.721}
SPL {X  -153.385, Y  +325.878, Z    +0.000, E1   +53.068, E3 +281641.302}
SPL {X  -151.310, Y  +320.369, Z    +0.000, E1   +52.706, E3 +281651.501}
SPL {X  -148.923, Y  +314.679, Z    +0.000, E1   +52.172, E3 +281662.585}
SPL {X  -146.846, Y  +310.168, Z    +0.000, E1   +51.697, E3 +281671.646}
SPL {X  -140.627, Y  +298.437, Z    +0.000, E1   +54.251, E3 +281675.905}
SPL {X  -122.064, Y  +272.747, Z    +0.000, E1   +48.156, E3 +281781.431}
ENDSPLINE

SPLINE
SPL {X  -148.173, Y  +313.009, Z    +0.000, E1   +35.624, E3 +281864.476}
SPL {X  -159.343, Y  +347.032, Z    +0.000, E1   +21.245, E3 +281868.320}
SPL {X  -162.355, Y  +368.197, Z    +0.000, E1    +9.799, E3 +281869.489}
SPL {X  -162.819, Y  +380.071, Z    +0.000, E1    +2.240, E3 +281869.483}
SPL {X  -162.820, Y  +383.414, Z    +0.000, E1    -0.499, E3 +281869.446}
SPL {X  -162.820, Y  +385.055, Z    +0.000, E1    -2.040, E3 +281869.090}
SPL {X  -162.820, Y  +388.271, Z    +0.000, E1    -5.458, E3 +281869.252}
SPL {X  -162.820, Y  +393.153, Z    +0.000, E1   -11.600, E3 +281869.129}
SPL {X  -162.820, Y  +400.748, Z    +0.000, E1   -21.791, E3 +281868.921}
SPL {X  -162.820, Y  +413.615, Z    +0.000, E1   -37.560, E3 +281869.015}
SPL {X  -162.820, Y  +456.390, Z    +0.000, E1   -57.415, E3 +281886.056}
SPL {X  -162.820, Y  +525.017, Z    +0.000, E1   -58.379, E3 +281956.721}
ENDSPLINE

SPLINE
SPL {X  -162.820, Y  +520.266, Z    +0.000, E1   -55.155, E3 +281971.213}
ENDSPLINE

SPLINE
SPL {X  -162.820, Y  +529.742, Z    +0.000, E1   -55.146, E3 +281984.929}
SPL {X  -162.820, Y  +538.383, Z    +0.000, E1   -55.306, E3 +281996.381}
SPL {X  -162.820, Y  +544.790, Z    +0.000, E1   -55.066, E3 +282007.182}
SPL {X  -162.820, Y  +552.981, Z    +0.000, E1   -55.286, E3 +282017.644}
SPL {X  -162.820, Y  +560.767, Z    +0.000, E1   -55.137, E3 +282029.953}
SPL {X  -162.820, Y  +570.590, Z    +0.000, E1   -55.270, E3 +282043.287}
SPL {X  -162.820, Y  +580.865, Z    +0.000, E1   -55.132, E3 +282059.243}
SPL {X  -162.820, Y  +591.604, Z    +0.000, E1   -55.202, E3 +282074.181}
SPL {X  -162.820, Y  +600.465, Z    +0.000, E1   -55.218, E3 +282086.969}
SPL {X  -162.820, Y  +609.951, Z    +0.000, E1   -55.211, E3 +282100.717}
SPL {X  -162.820, Y  +618.960, Z    +0.000, E1   -55.186, E3 +282113.937}
SPL {X  -162.820, Y  +627.322, Z    +0.000, E1   -55.201, E3 +282125.872}
SPL {X  -162.820, Y  +634.693, Z    +0.000, E1   -55.198, E3 +282136.589}
SPL {X  -162.820, Y  +642.452, Z    +0.000, E1   -55.141, E3 +282148.195}
SPL {X  -162.820, Y  +652.837, Z    +0.000, E1   -55.281, E3 +282162.463}
SPL {X  -162.820, Y  +660.849, Z    +0.000, E1   -55.101, E3 +282175.012}
SPL {X  -162.820, Y  +671.259, Z    +0.000, E1   -55.266, E3 +282189.308}
SPL {X  -162.498, Y  +683.731, Z    +0.000, E1   -55.157, E3 +282208.018}
SPL {X  -161.784, Y  +691.841, Z    +0.000, E1   -55.010, E3 +282220.474}
SPL {X  -161.070, Y  +697.305, Z    +0.000, E1   -54.828, E3 +282229.552}
SPL {X  -159.751, Y  +704.965, Z    +0.000, E1   -54.697, E3 +282241.538}
SPL {X  -158.271, Y  +711.718, Z    +0.000, E1   -54.504, E3 +282252.347}
SPL {X  -157.115, Y  +716.223, Z    +0.000, E1   -54.227, E3 +282260.538}
SPL {X  -155.622, Y  +721.376, Z    +0.000, E1   -53.849, E3 +282270.138}
SPL {X  -153.323, Y  +728.294, Z    +0.000, E1   -53.618, E3 +282281.611}
SPL {X  -150.606, Y  +735.372, Z    +0.000, E1   -53.091, E3 +282294.608}
SPL {X  -148.712, Y  +739.795, Z    +0.000, E1   -52.656, E3 +282303.171}
SPL {X  -146.885, Y  +743.751, Z    +0.000, E1   -52.544, E3 +282309.444}
SPL {X  -144.373, Y  +748.778, Z    +0.000, E1   -52.887, E3 +282314.907}
SPL {X  -137.947, Y  +759.993, Z    +0.000, E1   -55.381, E3 +282318.016}
SPL {X  -123.111, Y  +780.056, Z    +0.000, E1   -48.144, E3 +282417.152}
ENDSPLINE

SPLINE
SPL {X  -146.599, Y  +744.345, Z    +0.000, E1   -36.661, E3 +282502.155}
SPL {X  -157.185, Y  +715.965, Z    +0.000, E1   -25.340, E3 +282505.205}
SPL {X  -159.997, Y  +703.690, Z    +0.000, E1   -19.457, E3 +282506.533}
SPL {X  -161.886, Y  +690.913, Z    +0.000, E1   -12.672, E3 +282510.661}
SPL {X  -162.700, Y  +679.756, Z    +0.000, E1    -6.060, E3 +282509.871}
SPL {X  -162.820, Y  +673.439, Z    +0.000, E1    -1.797, E3 +282509.973}
SPL {X  -162.820, Y  +670.554, Z    +0.000, E1    +0.472, E3 +282509.505}
SPL {X  -162.820, Y  +667.789, Z    +0.000, E1    +3.144, E3 +282509.527}
SPL {X  -162.820, Y  +664.083, Z    +0.000, E1    +7.387, E3 +282509.418}
SPL {X  -162.820, Y  +659.344, Z    +0.000, E1   +13.535, E3 +282508.982}
SPL {X  -162.820, Y  +653.403, Z    +0.000, E1   +21.415, E3 +282509.397}
SPL {X  -162.820, Y  +642.162, Z    +0.000, E1   +35.510, E3 +282508.709}
SPL {X  -162.820, Y  +598.675, Z    +0.000, E1   +56.845, E3 +282526.022}
SPL {X  -162.820, Y  +543.175, Z    +0.000, E1   +54.504, E3 +282601.876}
SPL {X  -162.820, Y  +538.115, Z    +0.000, E1   +53.658, E3 +282614.927}
SPL {X  -162.820, Y  +527.429, Z    +0.000, E1   +53.760, E3 +282630.657}
SPL {X  -162.820, Y  +518.365, Z    +0.000, E1   +53.683, E3 +282644.915}
SPL {X  -162.820, Y  +508.465, Z    +0.000, E1   +53.706, E3 +282660.129}
SPL {X  -162.820, Y  +499.206, Z    +0.000, E1   +53.779, E3 +282673.569}
SPL {X  -162.820, Y  +493.008, Z    +0.000, E1   +53.586, E3 +282684.378}
SPL {X  -162.820, Y  +485.759, Z    +0.000, E1   +53.138, E3 +282698.385}
ENDSPLINE

SPLINE
SPL {X  -162.820, Y  +494.645, Z    +0.000, E1   +48.544, E3 +282710.861}
ENDSPLINE

SPLINE
SPL {X  -162.820, Y  +486.578, Z    +0.000, E1   +49.194, E3 +282721.657}
SPL {X  -162.820, Y  +476.731, Z    +0.000, E1   +50.039, E3 +282734.080}
SPL {X  -162.820, Y  +466.442, Z    +0.000, E1   +50.873, E3 +282746.749}
SPL {X  -162.820, Y  +455.624, Z    +0.000, E1   +51.698, E3 +282759.820}
SPL {X  -162.820, Y  +444.568, Z    +0.000, E1   +52.608, E3 +282772.133}
SPL {X  -162.820, Y  +432.435, Z    +0.000, E1   +53.605, E3 +282785.016}
SPL {X  -162.820, Y  +419.875, Z    +0.000, E1   +54.604, E3 +282797.690}
SPL {X  -162.820, Y  +414.181, Z    +0.000, E1   +54.446, E3 +282807.124}
SPL {X  -162.820, Y  +407.616, Z    +0.000, E1   +54.585, E3 +282815.958}
SPL {X  -162.820, Y  +400.244, Z    +0.000, E1   +54.630, E3 +282826.677}
SPL {X  -162.820, Y  +389.249, Z    +0.000, E1   +54.752, E3 +282842.256}
SPL {X  -162.799, Y  +377.862, Z    +0.000, E1   +54.622, E3 +282859.886}
SPL {X  -162.216, Y  +366.490, Z    +0.000, E1   +54.549, E3 +282877.182}
SPL {X  -160.880, Y  +355.442, Z    +0.000, E1   +54.372, E3 +282894.638}
SPL {X  -159.457, Y  +347.579, Z    +0.000, E1   +54.148, E3 +282907.375}
SPL {X  -158.033, Y  +341.310, Z    +0.000, E1   +53.819, E3 +282918.711}
SPL {X  -155.608, Y  +332.578, Z    +0.000, E1   +53.425, E3 +282933.983}
SPL {X  -152.785, Y  +324.223, Z    +0.000, E1   +52.975, E3 +282948.742}
SPL {X  -150.663, Y  +318.766, Z    +0.000, E1   +52.574, E3 +282958.775}
SPL {X  -148.923, Y  +314.679, Z    +0.000, E1   +52.172, E3 +282966.933}
SPL {X  -146.846, Y  +310.168, Z    +0.000, E1   +51.697, E3 +282975.994}
SPL {X  -140.627, Y  +298.437, Z    +0.000, E1   +54.251, E3 +282980.253}
SPL {X  -122.064, Y  +272.747, Z    +0.000, E1   +48.156, E3 +283085.779}
ENDSPLINE

SPLINE
SPL {X  -148.173, Y  +313.009, Z    +0.000, E1   +35.624, E3 +283168.824}
SPL {X  -158.289, Y  +342.356, Z    +0.000, E1   +23.452, E3 +283171.814}
SPL {X  -161.301, Y  +358.312, Z    +0.000, E1   +15.384, E3 +283173.771}
SPL {X  -162.692, Y  +374.052, Z    +0.000, E1    +6.208, E3 +283173.709}
SPL {X  -162.820, Y  +381.030, Z    +0.000, E1    +1.454, E3 +283173.888}
SPL {X  -162.820, Y  +384.274, Z    +0.000, E1    -1.205, E3 +283173.607}
SPL {X  -162.820, Y  +388.271, Z    +0.000, E1    -5.458, E3 +283173.600}
SPL {X  -162.820, Y  +394.827, Z    +0.000, E1   -13.677, E3 +283173.290}
SPL {X  -162.820, Y  +402.977, Z    +0.000, E1   -24.772, E3 +283173.572}
SPL {X  -162.820, Y  +413.615, Z    +0.000, E1   -37.560, E3 +283173.362}
SPL {X  -162.820, Y  +456.390, Z    +0.000, E1   -57.415, E3 +283190.404}
SPL {X  -162.820, Y  +525.017, Z    +0.000, E1   -58.379, E3 +283261.069}
ENDSPLINE

SPLINE
SPL {X  -162.820, Y  +515.796, Z    +0.000, E1   -54.952, E3 +283270.175}
ENDSPLINE

SPLINE
SPL {X  -162.820, Y  +522.537, Z    +0.000, E1   -55.218, E3 +283278.350}
SPL {X  -162.820, Y  +529.742, Z    +0.000, E1   -55.146, E3 +283289.277}
SPL {X  -162.820, Y  +538.383, Z    +0.000, E1   -55.306, E3 +283300.729}
SPL {X  -162.820, Y  +544.790, Z    +0.000, E1   -55.066, E3 +283311.530}
SPL {X  -162.820, Y  +552.981, Z    +0.000, E1   -55.286, E3 +283321.992}
SPL {X  -162.820, Y  +560.767, Z    +0.000, E1   -55.137, E3 +283334.300}
SPL {X  -162.820, Y  +570.590, Z    +0.000, E1   -55.270, E3 +283347.634}
SPL {X  -162.820, Y  +577.946, Z    +0.000, E1   -55.110, E3 +283359.272}
SPL {X  -162.820, Y  +583.981, Z    +0.000, E1   -55.057, E3 +283368.355}
SPL {X  -162.820, Y  +594.246, Z    +0.000, E1   -55.310, E3 +283381.790}
SPL {X  -162.820, Y  +601.811, Z    +0.000, E1   -55.027, E3 +283394.318}
SPL {X  -162.820, Y  +609.951, Z    +0.000, E1   -55.211, E3 +283405.064}
SPL {X  -162.820, Y  +617.278, Z    +0.000, E1   -55.256, E3 +283415.289}
SPL {X  -162.820, Y  +625.209, Z    +0.000, E1   -55.167, E3 +283427.480}
SPL {X  -162.820, Y  +634.693, Z    +0.000, E1   -55.198, E3 +283440.937}
SPL {X  -162.820, Y  +642.452, Z    +0.000, E1   -55.141, E3 +283452.543}
SPL {X  -162.820, Y  +652.837, Z    +0.000, E1   -55.281, E3 +283466.811}
SPL {X  -162.820, Y  +660.849, Z    +0.000, E1   -55.101, E3 +283479.360}
SPL {X  -162.820, Y  +668.534, Z    +0.000, E1   -55.182, E3 +283490.074}
SPL {X  -162.763, Y  +677.803, Z    +0.000, E1   -55.175, E3 +283503.580}
SPL {X  -162.314, Y  +686.325, Z    +0.000, E1   -55.173, E3 +283515.860}
SPL {X  -161.784, Y  +691.841, Z    +0.000, E1   -55.010, E3 +283524.822}
SPL {X  -160.705, Y  +699.660, Z    +0.000, E1   -54.830, E3 +283537.482}
SPL {X  -158.809, Y  +709.418, Z    +0.000, E1   -54.602, E3 +283552.954}
SPL {X  -157.115, Y  +716.223, Z    +0.000, E1   -54.227, E3 +283564.886}
SPL {X  -154.825, Y  +723.894, Z    +0.000, E1   -53.830, E3 +283578.426}
SPL {X  -152.160, Y  +731.445, Z    +0.000, E1   -53.336, E3 +283591.968}
SPL {X  -150.059, Y  +736.687, Z    +0.000, E1   -53.023, E3 +283601.134}
SPL {X  -147.746, Y  +741.922, Z    +0.000, E1   -52.631, E3 +283610.842}
SPL {X  -144.373, Y  +748.778, Z    +0.000, E1   -52.887, E3 +283619.255}
SPL {X  -137.947, Y  +759.993, Z    +0.000, E1   -55.381, E3 +283622.364}
SPL {X  -123.111, Y  +780.056, Z    +0.000, E1   -48.144, E3 +283721.500}
ENDSPLINE

SPLINE
SPL {X  -146.599, Y  +744.345, Z    +0.000, E1   -36.661, E3 +283806.503}
SPL {X  -158.886, Y  +709.076, Z    +0.000, E1   -22.176, E3 +283810.375}
SPL {X  -161.886, Y  +690.913, Z    +0.000, E1   -12.672, E3 +283815.009}
SPL {X  -162.573, Y  +682.458, Z    +0.000, E1    -7.683, E3 +283814.510}
SPL {X  -162.817, Y  +674.426, Z    +0.000, E1    -2.573, E3 +283814.228}
SPL {X  -162.820, Y  +670.554, Z    +0.000, E1    +0.472, E3 +283813.853}
SPL {X  -162.820, Y  +667.789, Z    +0.000, E1    +3.144, E3 +283813.874}
SPL {X  -162.820, Y  +664.083, Z    +0.000, E1    +7.387, E3 +283813.766}
SPL {X  -162.820, Y  +659.344, Z    +0.000, E1   +13.535, E3 +283813.330}
SPL {X  -162.820, Y  +653.403, Z    +0.000, E1   +21.415, E3 +283813.744}
SPL {X  -162.820, Y  +642.162, Z    +0.000, E1   +35.510, E3 +283813.057}
SPL {X  -162.820, Y  +598.675, Z    +0.000, E1   +56.845, E3 +283830.369}
SPL {X  -162.820, Y  +543.175, Z    +0.000, E1   +54.504, E3 +283906.224}
SPL {X  -162.820, Y  +538.115, Z    +0.000, E1   +53.658, E3 +283919.275}
SPL {X  -162.820, Y  +527.429, Z    +0.000, E1   +53.760, E3 +283935.005}
SPL {X  -162.820, Y  +518.365, Z    +0.000, E1   +53.683, E3 +283949.263}
SPL {X  -162.820, Y  +510.654, Z    +0.000, E1   +53.658, E3 +283961.262}
SPL {X  -162.820, Y  +501.304, Z    +0.000, E1   +53.758, E3 +283974.950}
SPL {X  -162.820, Y  +493.008, Z    +0.000, E1   +53.586, E3 +283988.726}
SPL {X  -162.820, Y  +485.759, Z    +0.000, E1   +53.138, E3 +284002.733}
ENDSPLINE

SPLINE
SPL {X  -162.820, Y  +494.645, Z    +0.000, E1   +48.544, E3 +284015.209}
ENDSPLINE

SPLINE
SPL {X  -162.820, Y  +483.544, Z    +0.000, E1   +49.458, E3 +284029.987}
SPL {X  -162.820, Y  +468.441, Z    +0.000, E1   +50.759, E3 +284048.489}
SPL {X  -162.820, Y  +455.624, Z    +0.000, E1   +51.698, E3 +284064.167}
SPL {X  -162.820, Y  +444.568, Z    +0.000, E1   +52.608, E3 +284076.480}
SPL {X  -162.820, Y  +432.435, Z    +0.000, E1   +53.605, E3 +284089.363}
SPL {X  -162.820, Y  +419.900, Z    +0.000, E1   +54.598, E3 +284102.038}
SPL {X  -162.820, Y  +411.092, Z    +0.000, E1   +54.552, E3 +284115.558}
SPL {X  -162.820, Y  +400.244, Z    +0.000, E1   +54.630, E3 +284131.025}
SPL {X  -162.820, Y  +389.249, Z    +0.000, E1   +54.752, E3 +284146.604}
SPL {X  -162.820, Y  +380.650, Z    +0.000, E1   +54.601, E3 +284160.048}
SPL {X  -162.727, Y  +374.992, Z    +0.000, E1   +54.549, E3 +284168.730}
SPL {X  -162.216, Y  +366.490, Z    +0.000, E1   +54.549, E3 +284181.530}
SPL {X  -161.062, Y  +356.641, Z    +0.000, E1   +54.440, E3 +284196.648}
SPL {X  -159.761, Y  +349.086, Z    +0.000, E1   +54.132, E3 +284209.669}
SPL {X  -158.033, Y  +341.310, Z    +0.000, E1   +53.819, E3 +284223.059}
SPL {X  -155.608, Y  +332.578, Z    +0.000, E1   +53.425, E3 +284238.330}
SPL {X  -153.385, Y  +325.878, Z    +0.000, E1   +53.068, E3 +284249.998}
SPL {X  -151.310, Y  +320.369, Z    +0.000, E1   +52.706, E3 +284260.196}
SPL {X  -148.923, Y  +314.679, Z    +0.000, E1   +52.172, E3 +284271.281}
SPL {X  -146.846, Y  +310.168, Z    +0.000, E1   +51.697, E3 +284280.342}
SPL {X  -140.627, Y  +298.437, Z    +0.000, E1   +54.251, E3 +284284.601}
SPL {X  -122.064, Y  +272.747, Z    +0.000, E1   +48.156, E3 +284390.126}
ENDSPLINE

SPLINE
SPL {X  -148.173, Y  +313.009, Z    +0.000, E1   +35.624, E3 +284473.172}
SPL {X  -159.343, Y  +347.032, Z    +0.000, E1   +21.245, E3 +284477.015}
SPL {X  -161.787, Y  +362.186, Z    +0.000, E1   +13.182, E3 +284478.211}
SPL {X  -162.692, Y  +374.052, Z    +0.000, E1    +6.208, E3 +284478.057}
SPL {X  -162.820, Y  +382.143, Z    +0.000, E1    +0.693, E3 +284478.192}
SPL {X  -162.820, Y  +385.055, Z    +0.000, E1    -2.040, E3 +284477.786}
SPL {X  -162.820, Y  +388.271, Z    +0.000, E1    -5.458, E3 +284477.948}
SPL {X  -162.820, Y  +393.153, Z    +0.000, E1   -11.600, E3 +284477.825}
SPL {X  -162.820, Y  +400.748, Z    +0.000, E1   -21.791, E3 +284477.616}
SPL {X  -162.820, Y  +413.615, Z    +0.000, E1   -37.560, E3 +284477.710}
SPL {X  -162.820, Y  +452.521, Z    +0.000, E1   -56.942, E3 +284492.002}
SPL {X  -162.820, Y  +459.967, Z    +0.000, E1   -57.801, E3 +284497.298}
SPL {X  -162.820, Y  +525.017, Z    +0.000, E1   -58.379, E3 +284565.416}
ENDSPLINE

SPLINE
SPL {X  -162.820, Y  +520.266, Z    +0.000, E1   -55.155, E3 +284579.909}
ENDSPLINE

SPLINE
SPL {X  -162.820, Y  +529.742, Z    +0.000, E1   -55.146, E3 +284593.625}
SPL {X  -162.820, Y  +538.383, Z    +0.000, E1   -55.306, E3 +284605.077}
SPL {X  -162.820, Y  +544.790, Z    +0.000, E1   -55.066, E3 +284615.877}
SPL {X  -162.820, Y  +555.105, Z    +0.000, E1   -55.222, E3 +284629.998}
SPL {X  -162.820, Y  +563.355, Z    +0.000, E1   -55.172, E3 +284642.064}
SPL {X  -162.820, Y  +570.590, Z    +0.000, E1   -55.270, E3 +284651.982}
SPL {X  -162.820, Y  +580.865, Z    +0.000, E1   -55.132, E3 +284667.939}
SPL {X  -162.820, Y  +594.246, Z    +0.000, E1   -55.310, E3 +284686.138}
SPL {X  -162.820, Y  +601.811, Z    +0.000, E1   -55.027, E3 +284698.666}
SPL {X  -162.820, Y  +609.951, Z    +0.000, E1   -55.211, E3 +284709.412}
SPL {X  -162.820, Y  +618.960, Z    +0.000, E1   -55.186, E3 +284722.632}
SPL {X  -162.820, Y  +627.322, Z    +0.000, E1   -55.201, E3 +284734.568}
SPL {X  -162.820, Y  +634.693, Z    +0.000, E1   -55.198, E3 +284745.284}
SPL {X  -162.820, Y  +642.452, Z    +0.000, E1   -55.141, E3 +284756.891}
SPL {X  -162.820, Y  +649.370, Z    +0.000, E1   -55.160, E3 +284766.748}
SPL {X  -162.820, Y  +658.542, Z    +0.000, E1   -55.251, E3 +284779.626}
SPL {X  -162.820, Y  +671.259, Z    +0.000, E1   -55.266, E3 +284798.003}
SPL {X  -162.498, Y  +683.731, Z    +0.000, E1   -55.157, E3 +284816.713}
SPL {X  -161.784, Y  +691.841, Z    +0.000, E1   -55.010, E3 +284829.170}
SPL {X  -161.070, Y  +697.305, Z    +0.000, E1   -54.828, E3 +284838.248}
SPL {X  -159.751, Y  +704.965, Z    +0.000, E1   -54.697, E3 +284850.234}
SPL {X  -158.271, Y  +711.718, Z    +0.000, E1   -54.504, E3 +284861.042}
SPL {X  -157.115, Y  +716.223, Z    +0.000, E1   -54.227, E3 +284869.234}
SPL {X  -154.825, Y  +723.894, Z    +0.000, E1   -53.830, E3 +284882.774}
SPL {X  -152.160, Y  +731.445, Z    +0.000, E1   -53.336, E3 +284896.316}
SPL {X  -150.059, Y  +736.687, Z    +0.000, E1   -53.023, E3 +284905.482}
SPL {X  -147.746, Y  +741.922, Z    +0.000, E1   -52.631, E3 +284915.189}
SPL {X  -144.373, Y  +748.778, Z    +0.000, E1   -52.887, E3 +284923.602}
SPL {X  -137.947, Y  +759.993, Z    +0.000, E1   -55.381, E3 +284926.712}
SPL {X  -123.111, Y  +780.056, Z    +0.000, E1   -48.144, E3 +285025.848}
ENDSPLINE

SPLINE
SPL {X  -146.599, Y  +744.345, Z    +0.000, E1   -36.661, E3 +285110.851}
SPL {X  -157.185, Y  +715.965, Z    +0.000, E1   -25.340, E3 +285113.901}
SPL {X  -159.997, Y  +703.690, Z    +0.000, E1   -19.457, E3 +285115.229}
SPL {X  -161.886, Y  +690.913, Z    +0.000, E1   -12.672, E3 +285119.357}
SPL {X  -162.700, Y  +679.756, Z    +0.000, E1    -6.060, E3 +285118.566}
SPL {X  -162.820, Y  +673.439, Z    +0.000, E1    -1.797, E3 +285118.668}
SPL {X  -162.820, Y  +670.554, Z    +0.000, E1    +0.472, E3 +285118.201}
SPL {X  -162.820, Y  +667.789, Z    +0.000, E1    +3.144, E3 +285118.222}
SPL {X  -162.820, Y  +664.083, Z    +0.000, E1    +7.387, E3 +285118.114}
SPL {X  -162.820, Y  +659.344, Z    +0.000, E1   +13.535, E3 +285117.678}
SPL {X  -162.820, Y  +653.403, Z    +0.000, E1   +21.415, E3 +285118.092}
SPL {X  -162.820, Y  +642.162, Z    +0.000, E1   +35.510, E3 +285117.405}
SPL {X  -162.820, Y  +598.675, Z    +0.000, E1   +56.845, E3 +285134.717}
SPL {X  -162.820, Y  +542.287, Z    +0.000, E1   +54.257, E3 +285213.621}
SPL {X  -162.820, Y  +533.839, Z    +0.000, E1   +53.682, E3 +285230.042}
SPL {X  -162.820, Y  +525.300, Z    +0.000, E1   +53.701, E3 +285242.817}
SPL {X  -162.820, Y  +518.365, Z    +0.000, E1   +53.683, E3 +285253.611}
SPL {X  -162.820, Y  +510.654, Z    +0.000, E1   +53.658, E3 +285265.610}
SPL {X  -162.820, Y  +501.304, Z    +0.000, E1   +53.758, E3 +285279.298}
SPL {X  -162.820, Y  +493.008, Z    +0.000, E1   +53.586, E3 +285293.073}
SPL {X  -162.820, Y  +485.759, Z    +0.000, E1   +53.138, E3 +285307.081}
ENDSPLINE

SPLINE
SPL {X  -162.820, Y  +494.645, Z    +0.000, E1   +48.544, E3 +285319.557}
ENDSPLINE

SPLINE
SPL {X  -162.820, Y  +486.578, Z    +0.000, E1   +49.194, E3 +285330.353}
SPL {X  -162.820, Y  +476.731, Z    +0.000, E1   +50.039, E3 +285342.776}
SPL {X  -162.820, Y  +466.442, Z    +0.000, E1   +50.873, E3 +285355.444}
SPL {X  -162.820, Y  +455.624, Z    +0.000, E1   +51.698, E3 +285368.515}
SPL {X  -162.820, Y  +444.568, Z    +0.000, E1   +52.608, E3 +285380.828}
SPL {X  -162.820, Y  +432.435, Z    +0.000, E1   +53.605, E3 +285393.711}
SPL {X  -162.820, Y  +419.900, Z    +0.000, E1   +54.598, E3 +285406.386}
SPL {X  -162.820, Y  +411.092, Z    +0.000, E1   +54.552, E3 +285419.906}
SPL {X  -162.820, Y  +400.244, Z    +0.000, E1   +54.630, E3 +285435.372}
SPL {X  -162.820, Y  +389.249, Z    +0.000, E1   +54.752, E3 +285450.951}
SPL {X  -162.799, Y  +377.862, Z    +0.000, E1   +54.622, E3 +285468.582}
SPL {X  -162.373, Y  +368.447, Z    +0.000, E1   +54.597, E3 +285482.511}
SPL {X  -161.939, Y  +363.587, Z    +0.000, E1   +54.355, E3 +285491.123}
SPL {X  -161.062, Y  +356.641, Z    +0.000, E1   +54.440, E3 +285500.996}
SPL {X  -159.761, Y  +349.086, Z    +0.000, E1   +54.132, E3 +285514.017}
SPL {X  -158.451, Y  +343.033, Z    +0.000, E1   +53.828, E3 +285524.693}
SPL {X  -156.619, Y  +335.993, Z    +0.000, E1   +53.639, E3 +285536.340}
SPL {X  -154.959, Y  +330.520, Z    +0.000, E1   +53.198, E3 +285546.765}
SPL {X  -153.385, Y  +325.878, Z    +0.000, E1   +53.068, E3 +285554.346}
SPL {X  -151.310, Y  +320.369, Z    +0.000, E1   +52.706, E3 +285564.544}
SPL {X  -148.923, Y  +314.679, Z    +0.000, E1   +52.172, E3 +285575.629}
SPL {X  -146.846, Y  +310.168, Z    +0.000, E1   +51.697, E3 +285584.690}
SPL {X  -140.627, Y  +298.437, Z    +0.000, E1   +54.251, E3 +285588.949}
SPL {X  -122.064, Y  +272.747, Z    +0.000, E1   +48.156, E3 +285694.474}
ENDSPLINE

SPLINE
SPL {X  -148.173, Y  +313.009, Z    +0.000, E1   +35.624, E3 +285777.520}
SPL {X  -159.343, Y  +347.032, Z    +0.000, E1   +21.245, E3 +285781.363}
SPL {X  -162.355, Y  +368.197, Z    +0.000, E1    +9.799, E3 +285782.532}
SPL {X  -162.819, Y  +380.071, Z    +0.000, E1    +2.240, E3 +285782.527}
SPL {X  -162.820, Y  +383.414, Z    +0.000, E1    -0.499, E3 +285782.490}
SPL {X  -162.820, Y  +385.887, Z    +0.000, E1    -2.819, E3 +285782.212}
SPL {X  -162.820, Y  +389.383, Z    +0.000, E1    -6.871, E3 +285782.279}
SPL {X  -162.820, Y  +393.153, Z    +0.000, E1   -11.600, E3 +285782.172}
SPL {X  -162.820, Y  +400.748, Z    +0.000, E1   -21.791, E3 +285781.964}
SPL {X  -162.820, Y  +413.615, Z    +0.000, E1   -37.560, E3 +285782.058}
SPL {X  -162.820, Y  +456.390, Z    +0.000, E1   -57.415, E3 +285799.099}
SPL {X  -162.820, Y  +525.017, Z    +0.000, E1   -58.379, E3 +285869.764}
ENDSPLINE

SPLINE
SPL {X  -162.820, Y  +520.266, Z    +0.000, E1   -55.155, E3 +285884.257}
ENDSPLINE

SPLINE
SPL {X  -162.820, Y  +529.742, Z    +0.000, E1   -55.146, E3 +285897.973}
SPL {X  -162.820, Y  +538.383, Z    +0.000, E1   -55.306, E3 +285909.425}
SPL {X  -162.820, Y  +544.790, Z    +0.000, E1   -55.066, E3 +285920.225}
SPL {X  -162.820, Y  +552.981, Z    +0.000, E1   -55.286, E3 +285930.688}
SPL {X  -162.820, Y  +560.767, Z    +0.000, E1   -55.137, E3 +285942.996}
SPL {X  -162.820, Y  +570.590, Z    +0.000, E1   -55.270, E3 +285956.330}
SPL {X  -162.820, Y  +577.946, Z    +0.000, E1   -55.110, E3 +285967.968}
SPL {X  -162.820, Y  +583.981, Z    +0.000, E1   -55.057, E3 +285977.050}
SPL {X  -162.820, Y  +594.246, Z    +0.000, E1   -55.310, E3 +285990.486}
SPL {X  -162.820, Y  +601.811, Z    +0.000, E1   -55.027, E3 +286003.014}
SPL {X  -162.820, Y  +609.951, Z    +0.000, E1   -55.211, E3 +286013.760}
SPL {X  -162.820, Y  +618.960, Z    +0.000, E1   -55.186, E3 +286026.980}
SPL {X  -162.820, Y  +627.322, Z    +0.000, E1   -55.201, E3 +286038.916}
SPL {X  -162.820, Y  +634.693, Z    +0.000, E1   -55.198, E3 +286049.632}
SPL {X  -162.820, Y  +642.452, Z    +0.000, E1   -55.141, E3 +286061.239}
SPL {X  -162.820, Y  +652.837, Z    +0.000, E1   -55.281, E3 +286075.507}
SPL {X  -162.820, Y  +660.849, Z    +0.000, E1   -55.101, E3 +286088.056}
SPL {X  -162.820, Y  +668.534, Z    +0.000, E1   -55.182, E3 +286098.769}
SPL {X  -162.763, Y  +677.803, Z    +0.000, E1   -55.175, E3 +286112.275}
SPL {X  -162.084, Y  +688.960, Z    +0.000, E1   -55.150, E3 +286128.730}
SPL {X  -161.070, Y  +697.305, Z    +0.000, E1   -54.828, E3 +286142.595}
SPL {X  -159.751, Y  +704.965, Z    +0.000, E1   -54.697, E3 +286154.582}
SPL {X  -158.271, Y  +711.718, Z    +0.000, E1   -54.504, E3 +286165.390}
SPL {X  -157.115, Y  +716.223, Z    +0.000, E1   -54.227, E3 +286173.582}
SPL {X  -155.622, Y  +721.376, Z    +0.000, E1   -53.849, E3 +286183.182}
SPL {X  -153.323, Y  +728.294, Z    +0.000, E1   -53.618, E3 +286194.655}
SPL {X  -150.606, Y  +735.372, Z    +0.000, E1   -53.091, E3 +286207.652}
SPL {X  -148.712, Y  +739.795, Z    +0.000, E1   -52.656, E3 +286216.214}
SPL {X  -146.885, Y  +743.751, Z    +0.000, E1   -52.544, E3 +286222.488}
SPL {X  -144.373, Y  +748.778, Z    +0.000, E1   -52.887, E3 +286227.950}
SPL {X  -137.947, Y  +759.993, Z    +0.000, E1   -55.381, E3 +286231.060}
SPL {X  -123.111, Y  +780.056, Z    +0.000, E1   -48.144, E3 +286330.195}
ENDSPLINE

SPLINE
SPL {X  -146.599, Y  +744.345, Z    +0.000, E1   -36.661, E3 +286415.199}
SPL {X  -158.886, Y  +709.076, Z    +0.000, E1   -22.176, E3 +286419.071}
SPL {X  -161.886, Y  +690.913, Z    +0.000, E1   -12.672, E3 +286423.705}
SPL {X  -162.573, Y  +682.458, Z    +0.000, E1    -7.683, E3 +286423.206}
SPL {X  -162.817, Y  +674.426, Z    +0.000, E1    -2.573, E3 +286422.924}
SPL {X  -162.820, Y  +670.554, Z    +0.000, E1    +0.472, E3 +286422.548}
SPL {X  -162.820, Y  +667.789, Z    +0.000, E1    +3.144, E3 +286422.570}
SPL {X  -162.820, Y  +664.083, Z    +0.000, E1    +7.387, E3 +286422.462}
SPL {X  -162.820, Y  +659.344, Z    +0.000, E1   +13.535, E3 +286422.025}
SPL {X  -162.820, Y  +653.403, Z    +0.000, E1   +21.415, E3 +286422.440}
SPL {X  -162.820, Y  +642.162, Z    +0.000, E1   +35.510, E3 +286421.753}
SPL {X  -162.820, Y  +598.675, Z    +0.000, E1   +56.845, E3 +286439.065}
SPL {X  -162.820, Y  +543.175, Z    +0.000, E1   +54.504, E3 +286514.919}
SPL {X  -162.820, Y  +538.115, Z    +0.000, E1   +53.658, E3 +286527.971}
SPL {X  -162.820, Y  +527.429, Z    +0.000, E1   +53.760, E3 +286543.701}
SPL {X  -162.820, Y  +518.365, Z    +0.000, E1   +53.683, E3 +286557.958}
SPL {X  -162.820, Y  +510.654, Z    +0.000, E1   +53.658, E3 +286569.957}
SPL {X  -162.820, Y  +501.304, Z    +0.000, E1   +53.758, E3 +286583.646}
SPL {X  -162.820, Y  +493.008, Z    +0.000, E1   +53.586, E3 +286597.421}
SPL {X  -162.820, Y  +484.615, Z    +0.000, E1   +53.726, E3 +286609.352}
ENDSPLINE

SPLINE
SPL {X  -162.820, Y  +492.996, Z    +0.000, E1   +49.430, E3 +286621.898}
ENDSPLINE

SPLINE
SPL {X  -162.820, Y  +486.578, Z    +0.000, E1   +49.194, E3 +286634.701}
SPL {X  -162.820, Y  +476.731, Z    +0.000, E1   +50.039, E3 +286647.124}
SPL {X  -162.820, Y  +466.442, Z    +0.000, E1   +50.873, E3 +286659.792}
SPL {X  -162.820, Y  +455.624, Z    +0.000, E1   +51.698, E3 +286672.863}
SPL {X  -162.820, Y  +444.568, Z    +0.000, E1   +52.608, E3 +286685.176}
SPL {X  -162.820, Y  +432.435, Z    +0.000, E1   +53.605, E3 +286698.059}
SPL {X  -162.820, Y  +419.900, Z    +0.000, E1   +54.598, E3 +286710.734}
SPL {X  -162.820, Y  +411.092, Z    +0.000, E1   +54.552, E3 +286724.254}
SPL {X  -162.820, Y  +400.244, Z    +0.000, E1   +54.630, E3 +286739.720}
SPL {X  -162.820, Y  +389.249, Z    +0.000, E1   +54.752, E3 +286755.299}
SPL {X  -162.820, Y  +380.650, Z    +0.000, E1   +54.601, E3 +286768.744}
SPL {X  -162.727, Y  +374.992, Z    +0.000, E1   +54.549, E3 +286777.426}
SPL {X  -162.216, Y  +366.490, Z    +0.000, E1   +54.549, E3 +286790.225}
SPL {X  -161.062, Y  +356.641, Z    +0.000, E1   +54.440, E3 +286805.343}
SPL {X  -159.761, Y  +349.086, Z    +0.000, E1   +54.132, E3 +286818.365}
SPL {X  -158.033, Y  +341.310, Z    +0.000, E1   +53.819, E3 +286831.755}
SPL {X  -156.195, Y  +334.528, Z    +0.000, E1   +53.534, E3 +286843.320}
SPL {X  -154.120, Y  +327.988, Z    +0.000, E1   +53.171, E3 +286855.177}
SPL {X  -151.310, Y  +320.369, Z    +0.000, E1   +52.706, E3 +286868.892}
SPL {X  -148.923, Y  +314.679, Z    +0.000, E1   +52.172, E3 +286879.977}
SPL {X  -146.846, Y  +310.168, Z    +0.000, E1   +51.697, E3 +286889.038}
SPL {X  -140.627, Y  +298.437, Z    +0.000, E1   +54.251, E3 +286893.297}
SPL {X  -122.064, Y  +272.747, Z    +0.000, E1   +48.156, E3 +286998.822}
ENDSPLINE

SPLINE
SPL {X  -148.173, Y  +313.009, Z    +0.000, E1   +35.624, E3 +287081.867}
SPL {X  -158.289, Y  +342.356, Z    +0.000, E1   +23.452, E3 +287084.857}
SPL {X  -161.301, Y  +358.312, Z    +0.000, E1   +15.384, E3 +287086.815}
SPL {X  -162.692, Y  +374.052, Z    +0.000, E1    +6.208, E3 +287086.753}
SPL {X  -162.820, Y  +381.030, Z    +0.000, E1    +1.454, E3 +287086.932}
SPL {X  -162.820, Y  +384.274, Z    +0.000, E1    -1.205, E3 +287086.651}
SPL {X  -162.820, Y  +388.271, Z    +0.000, E1    -5.458, E3 +287086.643}
SPL {X  -162.820, Y  +394.827, Z    +0.000, E1   -13.677, E3 +287086.333}
SPL {X  -162.820, Y  +402.977, Z    +0.000, E1   -24.772, E3 +287086.615}
SPL {X  -162.820, Y  +413.615, Z    +0.000, E1   -37.560, E3 +287086.406}
SPL {X  -162.820, Y  +456.390, Z    +0.000, E1   -57.415, E3 +287103.447}
SPL {X  -162.820, Y  +525.017, Z    +0.000, E1   -58.379, E3 +287174.112}
ENDSPLINE

SPLINE
SPL {X  -162.820, Y  +515.796, Z    +0.000, E1   -54.952, E3 +287183.219}
ENDSPLINE

SPLINE
SPL {X  -162.820, Y  +522.537, Z    +0.000, E1   -55.218, E3 +287191.394}
SPL {X  -162.820, Y  +529.742, Z    +0.000, E1   -55.146, E3 +287202.321}
SPL {X  -162.820, Y  +538.383, Z    +0.000, E1   -55.306, E3 +287213.773}
SPL {X  -162.820, Y  +544.790, Z    +0.000, E1   -55.066, E3 +287224.573}
SPL {X  -162.820, Y  +552.981, Z    +0.000, E1   -55.286, E3 +287235.035}
SPL {X  -162.820, Y  +560.767, Z    +0.000, E1   -55.137, E3 +287247.344}
SPL {X  -162.820, Y  +570.590, Z    +0.000, E1   -55.270, E3 +287260.678}
SPL {X  -162.820, Y  +577.946, Z    +0.000, E1   -55.110, E3 +287272.316}
SPL {X  -162.820, Y  +583.981, Z    +0.000, E1   -55.057, E3 +287281.398}
SPL {X  -162.820, Y  +591.604, Z    +0.000, E1   -55.202, E3 +287291.572}
SPL {X  -162.820, Y  +600.465, Z    +0.000, E1   -55.218, E3 +287304.360}
SPL {X  -162.820, Y  +609.951, Z    +0.000, E1   -55.211, E3 +287318.108}
SPL {X  -162.820, Y  +617.278, Z    +0.000, E1   -55.256, E3 +287328.332}
SPL {X  -162.820, Y  +625.209, Z    +0.000, E1   -55.167, E3 +287340.524}
SPL {X  -162.820, Y  +634.693, Z    +0.000, E1   -55.198, E3 +287353.980}
SPL {X  -162.820, Y  +642.452, Z    +0.000, E1   -55.141, E3 +287365.587}
SPL {X  -162.820, Y  +652.837, Z    +0.000, E1   -55.281, E3 +287379.855}
SPL {X  -162.820, Y  +660.849, Z    +0.000, E1   -55.101, E3 +287392.403}
SPL {X  -162.820, Y  +668.534, Z    +0.000, E1   -55.182, E3 +287403.117}
SPL {X  -162.763, Y  +677.803, Z    +0.000, E1   -55.175, E3 +287416.623}
SPL {X  -162.314, Y  +686.325, Z    +0.000, E1   -55.173, E3 +287428.903}
SPL {X  -161.784, Y  +691.841, Z    +0.000, E1   -55.010, E3 +287437.865}
SPL {X  -161.070, Y  +697.305, Z    +0.000, E1   -54.828, E3 +287446.943}
SPL {X  -159.751, Y  +704.965, Z    +0.000, E1   -54.697, E3 +287458.929}
SPL {X  -158.271, Y  +711.718, Z    +0.000, E1   -54.504, E3 +287469.738}
SPL {X  -157.115, Y  +716.223, Z    +0.000, E1   -54.227, E3 +287477.930}
SPL {X  -155.622, Y  +721.376, Z    +0.000, E1   -53.849, E3 +287487.530}
SPL {X  -153.323, Y  +728.294, Z    +0.000, E1   -53.618, E3 +287499.003}
SPL {X  -150.606, Y  +735.372, Z    +0.000, E1   -53.091, E3 +287511.999}
SPL {X  -148.712, Y  +739.795, Z    +0.000, E1   -52.656, E3 +287520.562}
SPL {X  -146.885, Y  +743.751, Z    +0.000, E1   -52.544, E3 +287526.835}
SPL {X  -144.373, Y  +748.778, Z    +0.000, E1   -52.887, E3 +287532.298}
SPL {X  -137.947, Y  +759.993, Z    +0.000, E1   -55.381, E3 +287535.408}
SPL {X  -123.111, Y  +780.056, Z    +0.000, E1   -48.144, E3 +287634.543}
ENDSPLINE

SPLINE
SPL {X  -146.599, Y  +744.345, Z    +0.000, E1   -36.661, E3 +287719.547}
SPL {X  -158.886, Y  +709.076, Z    +0.000, E1   -22.176, E3 +287723.419}
SPL {X  -161.886, Y  +690.913, Z    +0.000, E1   -12.672, E3 +287728.053}
SPL {X  -162.573, Y  +682.458, Z    +0.000, E1    -7.683, E3 +287727.554}
SPL {X  -162.817, Y  +674.426, Z    +0.000, E1    -2.573, E3 +287727.272}
SPL {X  -162.820, Y  +670.554, Z    +0.000, E1    +0.472, E3 +287726.896}
SPL {X  -162.820, Y  +667.789, Z    +0.000, E1    +3.144, E3 +287726.918}
SPL {X  -162.820, Y  +664.083, Z    +0.000, E1    +7.387, E3 +287726.810}
SPL {X  -162.820, Y  +659.344, Z    +0.000, E1   +13.535, E3 +287726.373}
SPL {X  -162.820, Y  +653.403, Z    +0.000, E1   +21.415, E3 +287726.788}
SPL {X  -162.820, Y  +642.162, Z    +0.000, E1   +35.510, E3 +287726.100}
SPL {X  -162.820, Y  +598.675, Z    +0.000, E1   +56.845, E3 +287743.413}
SPL {X  -162.820, Y  +543.175, Z    +0.000, E1   +54.504, E3 +287819.267}
SPL {X  -162.820, Y  +538.115, Z    +0.000, E1   +53.658, E3 +287832.319}
SPL {X  -162.820, Y  +527.429, Z    +0.000, E1   +53.760, E3 +287848.048}
SPL {X  -162.820, Y  +518.365, Z    +0.000, E1   +53.683, E3 +287862.306}
SPL {X  -162.820, Y  +510.654, Z    +0.000, E1   +53.658, E3 +287874.305}
SPL {X  -162.820, Y  +501.304, Z    +0.000, E1   +53.758, E3 +287887.994}
SPL {X  -162.820, Y  +493.008, Z    +0.000, E1   +53.586, E3 +287901.769}
SPL {X  -162.820, Y  +484.615, Z    +0.000, E1   +53.726, E3 +287913.700}
ENDSPLINE

SPLINE
SPL {X  -162.820, Y  +492.996, Z    +0.000, E1   +49.430, E3 +287926.246}
ENDSPLINE

SPLINE
SPL {X  -162.820, Y  +483.544, Z    +0.000, E1   +49.458, E3 +287943.030}
SPL {X  -162.820, Y  +468.441, Z    +0.000, E1   +50.759, E3 +287961.533}
SPL {X  -162.820, Y  +455.624, Z    +0.000, E1   +51.698, E3 +287977.211}
SPL {X  -162.820, Y  +444.568, Z    +0.000, E1   +52.608, E3 +287989.524}
SPL {X  -162.820, Y  +432.435, Z    +0.000, E1   +53.605, E3 +288002.407}
SPL {X  -162.820, Y  +419.900, Z    +0.000, E1   +54.598, E3 +288015.081}
SPL {X  -162.820, Y  +411.092, Z    +0.000, E1   +54.552, E3 +288028.601}
SPL {X  -162.820, Y  +400.244, Z    +0.000, E1   +54.630, E3 +288044.068}
SPL {X  -162.820, Y  +389.249, Z    +0.000, E1   +54.752, E3 +288059.647}
SPL {X  -162.820, Y  +380.650, Z    +0.000, E1   +54.601, E3 +288073.092}
SPL {X  -162.727, Y  +374.992, Z    +0.000, E1   +54.549, E3 +288081.774}
SPL {X  -162.373, Y  +368.447, Z    +0.000, E1   +54.597, E3 +288091.206}
SPL {X  -161.939, Y  +363.587, Z    +0.000, E1   +54.355, E3 +288099.818}
SPL {X  -161.062, Y  +356.641, Z    +0.000, E1   +54.440, E3 +288109.691}
SPL {X  -159.761, Y  +349.086, Z    +0.000, E1   +54.132, E3 +288122.712}
SPL {X  -158.033, Y  +341.310, Z    +0.000, E1   +53.819, E3 +288136.102}
SPL {X  -156.195, Y  +334.528, Z    +0.000, E1   +53.534, E3 +288147.668}
SPL {X  -154.120, Y  +327.988, Z    +0.000, E1   +53.171, E3 +288159.525}
SPL {X  -151.310, Y  +320.369, Z    +0.000, E1   +52.706, E3 +288173.240}
SPL {X  -148.923, Y  +314.679, Z    +0.000, E1   +52.172, E3 +288184.324}
SPL {X  -146.846, Y  +310.168, Z    +0.000, E1   +51.697, E3 +288193.386}
SPL {X  -140.627, Y  +298.437, Z    +0.000, E1   +54.251, E3 +288197.644}
SPL {X  -122.064, Y  +272.747, Z    +0.000, E1   +48.156, E3 +288303.170}
ENDSPLINE

SPLINE
SPL {X  -148.173, Y  +313.009, Z    +0.000, E1   +35.624, E3 +288386.215}
SPL {X  -159.343, Y  +347.032, Z    +0.000, E1   +21.245, E3 +288390.059}
SPL {X  -162.355, Y  +368.197, Z    +0.000, E1    +9.799, E3 +288391.228}
SPL {X  -162.819, Y  +380.071, Z    +0.000, E1    +2.240, E3 +288391.222}
SPL {X  -162.820, Y  +383.414, Z    +0.000, E1    -0.499, E3 +288391.185}
SPL {X  -162.820, Y  +385.887, Z    +0.000, E1    -2.819, E3 +288390.908}
SPL {X  -162.820, Y  +389.383, Z    +0.000, E1    -6.871, E3 +288390.975}
SPL {X  -162.820, Y  +393.153, Z    +0.000, E1   -11.600, E3 +288390.868}
SPL {X  -162.820, Y  +400.748, Z    +0.000, E1   -21.791, E3 +288390.660}
SPL {X  -162.820, Y  +413.615, Z    +0.000, E1   -37.560, E3 +288390.754}
SPL {X  -162.820, Y  +456.390, Z    +0.000, E1   -57.415, E3 +288407.795}
SPL {X  -162.820, Y  +525.017, Z    +0.000, E1   -58.379, E3 +288478.460}
ENDSPLINE

SPLINE
SPL {X  -162.820, Y  +520.266, Z    +0.000, E1   -55.155, E3 +288492.952}
ENDSPLINE

SPLINE
SPL {X  -162.820, Y  +529.742, Z    +0.000, E1   -55.146, E3 +288506.669}
SPL {X  -162.820, Y  +538.383, Z    +0.000, E1   -55.306, E3 +288518.121}
SPL {X  -162.820, Y  +544.790, Z    +0.000, E1   -55.066, E3 +288528.921}
SPL {X  -162.820, Y  +552.981, Z    +0.000, E1   -55.286, E3 +288539.383}
SPL {X  -162.820, Y  +560.767, Z    +0.000, E1   -55.137, E3 +288551.692}
SPL {X  -162.820, Y  +570.590, Z    +0.000, E1   -55.270, E3 +288565.026}
SPL {X  -162.820, Y  +577.946, Z    +0.000, E1   -55.110, E3 +288576.663}
SPL {X  -162.820, Y  +583.981, Z    +0.000, E1   -55.057, E3 +288585.746}
SPL {X  -162.820, Y  +594.246, Z    +0.000, E1   -55.310, E3 +288599.181}
SPL {X  -162.820, Y  +601.811, Z    +0.000, E1   -55.027, E3 +288611.709}
SPL {X  -162.820, Y  +609.951, Z    +0.000, E1   -55.211, E3 +288622.456}
SPL {X  -162.820, Y  +618.960, Z    +0.000, E1   -55.186, E3 +288635.676}
SPL {X  -162.820, Y  +627.322, Z    +0.000, E1   -55.201, E3 +288647.611}
SPL {X  -162.820, Y  +634.693, Z    +0.000, E1   -55.198, E3 +288658.328}
SPL {X  -162.820, Y  +642.452, Z    +0.000, E1   -55.141, E3 +288669.934}
SPL {X  -162.820, Y  +652.837, Z    +0.000, E1   -55.281, E3 +288684.202}
SPL {X  -162.820, Y  +660.849, Z    +0.000, E1   -55.101, E3 +288696.751}
SPL {X  -162.820, Y  +668.534, Z    +0.000, E1   -55.182, E3 +288707.465}
SPL {X  -162.763, Y  +677.803, Z    +0.000, E1   -55.175, E3 +288720.971}
SPL {X  -162.084, Y  +688.960, Z    +0.000, E1   -55.150, E3 +288737.426}
SPL {X  -161.070, Y  +697.305, Z    +0.000, E1   -54.828, E3 +288751.291}
SPL {X  -159.751, Y  +704.965, Z    +0.000, E1   -54.697, E3 +288763.277}
SPL {X  -158.271, Y  +711.718, Z    +0.000, E1   -54.504, E3 +288774.086}
SPL {X  -157.115, Y  +716.223, Z    +0.000, E1   -54.227, E3 +288782.277}
SPL {X  -155.622, Y  +721.376, Z    +0.000, E1   -53.849, E3 +288791.877}
SPL {X  -154.043, Y  +726.236, Z    +0.000, E1   -53.722, E3 +288799.626}
SPL {X  -152.160, Y  +731.445, Z    +0.000, E1   -53.336, E3 +288809.360}
SPL {X  -149.361, Y  +738.321, Z    +0.000, E1   -52.873, E3 +288821.822}
SPL {X  -145.628, Y  +746.320, Z    +0.000, E1   -52.740, E3 +288833.940}
SPL {X  -137.947, Y  +759.993, Z    +0.000, E1   -55.381, E3 +288839.755}
SPL {X  -123.111, Y  +780.056, Z    +0.000, E1   -48.144, E3 +288938.891}
ENDSPLINE

SPLINE
SPL {X  -146.599, Y  +744.345, Z    +0.000, E1   -36.661, E3 +289023.894}
SPL {X  -157.185, Y  +715.965, Z    +0.000, E1   -25.340, E3 +289026.944}
SPL {X  -159.997, Y  +703.690, Z    +0.000, E1   -19.457, E3 +289028.273}
SPL {X  -161.886, Y  +690.913, Z    +0.000, E1   -12.672, E3 +289032.401}
SPL {X  -162.700, Y  +679.756, Z    +0.000, E1    -6.060, E3 +289031.610}
SPL {X  -162.820, Y  +673.439, Z    +0.000, E1    -1.797, E3 +289031.712}
SPL {X  -162.820, Y  +670.554, Z    +0.000, E1    +0.472, E3 +289031.244}
SPL {X  -162.820, Y  +667.789, Z    +0.000, E1    +3.144, E3 +289031.266}
SPL {X  -162.820, Y  +664.083, Z    +0.000, E1    +7.387, E3 +289031.157}
SPL {X  -162.820, Y  +659.344, Z    +0.000, E1   +13.535, E3 +289030.721}
SPL {X  -162.820, Y  +653.403, Z    +0.000, E1   +21.415, E3 +289031.136}
SPL {X  -162.820, Y  +642.162, Z    +0.000, E1   +35.510, E3 +289030.448}
SPL {X  -162.820, Y  +598.675, Z    +0.000, E1   +56.845, E3 +289047.761}
SPL {X  -162.820, Y  +542.287, Z    +0.000, E1   +54.257, E3 +289126.664}
SPL {X  -162.820, Y  +533.839, Z    +0.000, E1   +53.682, E3 +289143.085}
SPL {X  -162.820, Y  +525.300, Z    +0.000, E1   +53.701, E3 +289155.860}
SPL {X  -162.820, Y  +518.365, Z    +0.000, E1   +53.683, E3 +289166.654}
SPL {X  -162.820, Y  +510.654, Z    +0.000, E1   +53.658, E3 +289178.653}
SPL {X  -162.820, Y  +501.304, Z    +0.000, E1   +53.758, E3 +289192.342}
SPL {X  -162.820, Y  +493.008, Z    +0.000, E1   +53.586, E3 +289206.117}
SPL {X  -162.820, Y  +485.759, Z    +0.000, E1   +53.138, E3 +289220.124}
ENDSPLINE

SPLINE
SPL {X  -162.820, Y  +494.645, Z    +0.000, E1   +48.544, E3 +289232.600}
ENDSPLINE

SPLINE
SPL {X  -162.820, Y  +486.578, Z    +0.000, E1   +49.194, E3 +289243.396}
SPL {X  -162.820, Y  +476.731, Z    +0.000, E1   +50.039, E3 +289255.819}
SPL {X  -162.820, Y  +466.442, Z    +0.000, E1   +50.873, E3 +289268.488}
SPL {X  -162.820, Y  +455.624, Z    +0.000, E1   +51.698, E3 +289281.559}
SPL {X  -162.820, Y  +444.568, Z    +0.000, E1   +52.608, E3 +289293.872}
SPL {X  -162.820, Y  +432.435, Z    +0.000, E1   +53.605, E3 +289306.755}
SPL {X  -162.820, Y  +419.875, Z    +0.000, E1   +54.604, E3 +289319.429}
SPL {X  -162.820, Y  +414.181, Z    +0.000, E1   +54.446, E3 +289328.863}
SPL {X  -162.820, Y  +407.616, Z    +0.000, E1   +54.585, E3 +289337.697}
SPL {X  -162.820, Y  +400.244, Z    +0.000, E1   +54.630, E3 +289348.416}
SPL {X  -162.820, Y  +389.249, Z    +0.000, E1   +54.752, E3 +289363.995}
SPL {X  -162.799, Y  +377.862, Z    +0.000, E1   +54.622, E3 +289381.625}
SPL {X  -162.373, Y  +368.447, Z    +0.000, E1   +54.597, E3 +289395.554}
SPL {X  -161.939, Y  +363.587, Z    +0.000, E1   +54.355, E3 +289404.166}
SPL {X  -161.062, Y  +356.641, Z    +0.000, E1   +54.440, E3 +289414.039}
SPL {X  -159.761, Y  +349.086, Z    +0.000, E1   +54.132, E3 +289427.060}
SPL {X  -158.451, Y  +343.033, Z    +0.000, E1   +53.828, E3 +289437.737}
SPL {X  -156.619, Y  +335.993, Z    +0.000, E1   +53.639, E3 +289449.383}
SPL {X  -154.959, Y  +330.520, Z    +0.000, E1   +53.198, E3 +289459.808}
SPL {X  -152.785, Y  +324.223, Z    +0.000, E1   +52.975, E3 +289470.481}
SPL {X  -150.663, Y  +318.766, Z    +0.000, E1   +52.574, E3 +289480.514}
SPL {X  -148.923, Y  +314.679, Z    +0.000, E1   +52.172, E3 +289488.672}
SPL {X  -146.846, Y  +310.168, Z    +0.000, E1   +51.697, E3 +289497.733}
SPL {X  -140.627, Y  +298.437, Z    +0.000, E1   +54.251, E3 +289501.992}
SPL {X  -122.064, Y  +272.747, Z    +0.000, E1   +48.156, E3 +289607.518}
ENDSPLINE

SPLINE
SPL {X  -143.204, Y  +303.021, Z    +0.000, E1   +38.944, E3 +289687.814}
SPL {X  -149.792, Y  +316.682, Z    +0.000, E1   +34.282, E3 +289691.392}
SPL {X  -159.343, Y  +347.032, Z    +0.000, E1   +21.245, E3 +289694.407}
SPL {X  -162.355, Y  +368.197, Z    +0.000, E1    +9.799, E3 +289695.576}
SPL {X  -162.819, Y  +380.071, Z    +0.000, E1    +2.240, E3 +289695.570}
SPL {X  -162.820, Y  +383.414, Z    +0.000, E1    -0.499, E3 +289695.533}
SPL {X  -162.820, Y  +385.055, Z    +0.000, E1    -2.040, E3 +289695.177}
SPL {X  -162.820, Y  +388.271, Z    +0.000, E1    -5.458, E3 +289695.339}
SPL {X  -162.820, Y  +394.827, Z    +0.000, E1   -13.677, E3 +289695.029}
SPL {X  -162.820, Y  +402.977, Z    +0.000, E1   -24.772, E3 +289695.311}
SPL {X  -162.820, Y  +413.615, Z    +0.000, E1   -37.560, E3 +289695.102}
SPL {X  -162.820, Y  +456.390, Z    +0.000, E1   -57.415, E3 +289712.143}
SPL {X  -162.820, Y  +525.017, Z    +0.000, E1   -58.379, E3 +289782.808}
ENDSPLINE

SPLINE
SPL {X  -162.820, Y  +515.796, Z    +0.000, E1   -54.952, E3 +289791.914}
ENDSPLINE

SPLINE
SPL {X  -162.820, Y  +522.537, Z    +0.000, E1   -55.218, E3 +289800.089}
SPL {X  -162.820, Y  +529.742, Z    +0.000, E1   -55.146, E3 +289811.016}
SPL {X  -162.820, Y  +538.383, Z    +0.000, E1   -55.306, E3 +289822.468}
SPL {X  -162.820, Y  +544.790, Z    +0.000, E1   -55.066, E3 +289833.269}
SPL {X  -162.820, Y  +552.981, Z    +0.000, E1   -55.286, E3 +289843.731}
SPL {X  -162.820, Y  +560.767, Z    +0.000, E1   -55.137, E3 +289856.040}
SPL {X  -162.820, Y  +570.590, Z    +0.000, E1   -55.270, E3 +289869.374}
SPL {X  -162.820, Y  +577.946, Z    +0.000, E1   -55.110, E3 +289881.011}
SPL {X  -162.820, Y  +583.981, Z    +0.000, E1   -55.057, E3 +289890.094}
SPL {X  -162.820, Y  +591.604, Z    +0.000, E1   -55.202, E3 +289900.268}
SPL {X  -162.820, Y  +600.465, Z    +0.000, E1   -55.218, E3 +289913.056}
SPL {X  -162.820, Y  +609.951, Z    +0.000, E1   -55.211, E3 +289926.804}
SPL {X  -162.820, Y  +617.278, Z    +0.000, E1   -55.256, E3 +289937.028}
SPL {X  -162.820, Y  +625.209, Z    +0.000, E1   -55.167, E3 +289949.220}
SPL {X  -162.820, Y  +634.693, Z    +0.000, E1   -55.198, E3 +289962.676}
SPL {X  -162.820, Y  +642.452, Z    +0.000, E1   -55.141, E3 +289974.282}
SPL {X  -162.820, Y  +652.837, Z    +0.000, E1   -55.281, E3 +289988.550}
SPL {X  -162.820, Y  +660.849, Z    +0.000, E1   -55.101, E3 +290001.099}
SPL {X  -162.820, Y  +668.534, Z    +0.000, E1   -55.182, E3 +290011.813}
SPL {X  -162.763, Y  +677.803, Z    +0.000, E1   -55.175, E3 +290025.319}
SPL {X  -162.314, Y  +686.325, Z    +0.000, E1   -55.173, E3 +290037.599}
SPL {X  -161.784, Y  +691.841, Z    +0.000, E1   -55.010, E3 +290046.561}
SPL {X  -161.070, Y  +697.305, Z    +0.000, E1   -54.828, E3 +290055.639}
SPL {X  -159.751, Y  +704.965, Z    +0.000, E1   -54.697, E3 +290067.625}
SPL {X  -158.271, Y  +711.718, Z    +0.000, E1   -54.504, E3 +290078.434}
SPL {X  -157.115, Y  +716.223, Z    +0.000, E1   -54.227, E3 +290086.625}
SPL {X  -154.825, Y  +723.894, Z    +0.000, E1   -53.830, E3 +290100.165}
SPL {X  -152.160, Y  +731.445, Z    +0.000, E1   -53.336, E3 +290113.708}
SPL {X  -149.361, Y  +738.321, Z    +0.000, E1   -52.873, E3 +290126.170}
SPL {X  -146.885, Y  +743.751, Z    +0.000, E1   -52.544, E3 +290135.531}
SPL {X  -144.373, Y  +748.778, Z    +0.000, E1   -52.887, E3 +290140.994}
SPL {X  -137.947, Y  +759.993, Z    +0.000, E1   -55.381, E3 +290144.103}
SPL {X  -123.111, Y  +780.056, Z    +0.000, E1   -48.144, E3 +290243.239}
ENDSPLINE

SPLINE
SPL {X  -146.599, Y  +744.345, Z    +0.000, E1   -36.661, E3 +290328.242}
SPL {X  -157.185, Y  +715.965, Z    +0.000, E1   -25.340, E3 +290331.292}
SPL {X  -159.997, Y  +703.690, Z    +0.000, E1   -19.457, E3 +290332.620}
SPL {X  -161.886, Y  +690.913, Z    +0.000, E1   -12.672, E3 +290336.748}
SPL {X  -162.700, Y  +679.756, Z    +0.000, E1    -6.060, E3 +290335.958}
SPL {X  -162.820, Y  +673.439, Z    +0.000, E1    -1.797, E3 +290336.060}
SPL {X  -162.820, Y  +670.554, Z    +0.000, E1    +0.472, E3 +290335.592}
SPL {X  -162.820, Y  +667.789, Z    +0.000, E1    +3.144, E3 +290335.614}
SPL {X  -162.820, Y  +664.083, Z    +0.000, E1    +7.387, E3 +290335.505}
SPL {X  -162.820, Y  +659.344, Z    +0.000, E1   +13.535, E3 +290335.069}
SPL {X  -162.820, Y  +653.403, Z    +0.000, E1   +21.415, E3 +290335.484}
SPL {X  -162.820, Y  +642.162, Z    +0.000, E1   +35.510, E3 +290334.796}
SPL {X  -162.820, Y  +598.675, Z    +0.000, E1   +56.845, E3 +290352.108}
SPL {X  -162.820, Y  +543.175, Z    +0.000, E1   +54.504, E3 +290427.963}
SPL {X  -162.820, Y  +538.115, Z    +0.000, E1   +53.658, E3 +290441.014}
SPL {X  -162.820, Y  +530.332, Z    +0.000, E1   +53.757, E3 +290452.157}
SPL {X  -162.820, Y  +525.300, Z    +0.000, E1   +53.701, E3 +290460.208}
SPL {X  -162.820, Y  +518.365, Z    +0.000, E1   +53.683, E3 +290471.002}
SPL {X  -162.820, Y  +510.654, Z    +0.000, E1   +53.658, E3 +290483.001}
SPL {X  -162.820, Y  +501.304, Z    +0.000, E1   +53.758, E3 +290496.689}
SPL {X  -162.820, Y  +493.008, Z    +0.000, E1   +53.586, E3 +290510.465}
SPL {X  -162.820, Y  +484.615, Z    +0.000, E1   +53.726, E3 +290522.395}
ENDSPLINE

SPLINE
SPL {X  -162.820, Y  +492.996, Z    +0.000, E1   +49.430, E3 +290534.941}
ENDSPLINE

SPLINE
SPL {X  -162.820, Y  +486.578, Z    +0.000, E1   +49.194, E3 +290547.744}
SPL {X  -162.820, Y  +476.731, Z    +0.000, E1   +50.039, E3 +290560.167}
SPL {X  -162.820, Y  +466.442, Z    +0.000, E1   +50.873, E3 +290572.835}
SPL {X  -162.820, Y  +455.624, Z    +0.000, E1   +51.698, E3 +290585.907}
SPL {X  -162.820, Y  +444.568, Z    +0.000, E1   +52.608, E3 +290598.219}
SPL {X  -162.820, Y  +432.435, Z    +0.000, E1   +53.605, E3 +290611.102}
SPL {X  -162.820, Y  +419.875, Z    +0.000, E1   +54.604, E3 +290623.777}
SPL {X  -162.820, Y  +414.181, Z    +0.000, E1   +54.446, E3 +290633.211}
SPL {X  -162.820, Y  +407.616, Z    +0.000, E1   +54.585, E3 +290642.045}
SPL {X  -162.820, Y  +400.244, Z    +0.000, E1   +54.630, E3 +290652.764}
SPL {X  -162.820, Y  +389.249, Z    +0.000, E1   +54.752, E3 +290668.343}
SPL {X  -162.820, Y  +380.650, Z    +0.000, E1   +54.601, E3 +290681.788}
SPL {X  -162.727, Y  +374.992, Z    +0.000, E1   +54.549, E3 +290690.470}
SPL {X  -162.373, Y  +368.447, Z    +0.000, E1   +54.597, E3 +290699.902}
SPL {X  -161.939, Y  +363.587, Z    +0.000, E1   +54.355, E3 +290708.514}
SPL {X  -161.062, Y  +356.641, Z    +0.000, E1   +54.440, E3 +290718.387}
SPL {X  -159.761, Y  +349.086, Z    +0.000, E1   +54.132, E3 +290731.408}
SPL {X  -158.451, Y  +343.033, Z    +0.000, E1   +53.828, E3 +290742.085}
SPL {X  -156.619, Y  +335.993, Z    +0.000, E1   +53.639, E3 +290753.731}
SPL {X  -154.959, Y  +330.520, Z    +0.000, E1   +53.198, E3 +290764.156}
SPL {X  -153.385, Y  +325.878, Z    +0.000, E1   +53.068, E3 +290771.737}
SPL {X  -151.310, Y  +320.369, Z    +0.000, E1   +52.706, E3 +290781.935}
SPL {X  -148.923, Y  +314.679, Z    +0.000, E1   +52.172, E3 +290793.020}
SPL {X  -146.846, Y  +310.168, Z    +0.000, E1   +51.697, E3 +290802.081}
SPL {X  -140.627, Y  +298.437, Z    +0.000, E1   +54.251, E3 +290806.340}
SPL {X  -122.064, Y  +272.747, Z    +0.000, E1   +48.156, E3 +290911.865}
ENDSPLINE

SPLINE
SPL {X  -148.173, Y  +313.009, Z    +0.000, E1   +35.624, E3 +290994.911}
SPL {X  -159.343, Y  +347.032, Z    +0.000, E1   +21.245, E3 +290998.755}
SPL {X  -162.355, Y  +368.197, Z    +0.000, E1    +9.799, E3 +290999.923}
SPL {X  -162.819, Y  +380.071, Z    +0.000, E1    +2.240, E3 +290999.918}
SPL {X  -162.820, Y  +383.414, Z    +0.000, E1    -0.499, E3 +290999.881}
SPL {X  -162.820, Y  +385.055, Z    +0.000, E1    -2.040, E3 +290999.525}
SPL {X  -162.820, Y  +388.271, Z    +0.000, E1    -5.458, E3 +290999.687}
SPL {X  -162.820, Y  +393.153, Z    +0.000, E1   -11.600, E3 +290999.564}
SPL {X  -162.820, Y  +400.748, Z    +0.000, E1   -21.791, E3 +290999.355}
SPL {X  -162.820, Y  +413.615, Z    +0.000, E1   -37.560, E3 +290999.449}
SPL {X  -162.820, Y  +456.390, Z    +0.000, E1   -57.415, E3 +291016.491}
SPL {X  -162.820, Y  +525.017, Z    +0.000, E1   -58.379, E3 +291087.156}
ENDSPLINE

SPLINE
SPL {X  -162.820, Y  +520.266, Z    +0.000, E1   -55.155, E3 +291101.648}
ENDSPLINE

SPLINE
SPL {X  -162.820, Y  +529.742, Z    +0.000, E1   -55.146, E3 +291115.364}
SPL {X  -162.820, Y  +538.383, Z    +0.000, E1   -55.306, E3 +291126.816}
SPL {X  -162.820, Y  +544.790, Z    +0.000, E1   -55.066, E3 +291137.616}
SPL {X  -162.820, Y  +552.981, Z    +0.000, E1   -55.286, E3 +291148.079}
SPL {X  -162.820, Y  +560.767, Z    +0.000, E1   -55.137, E3 +291160.387}
SPL {X  -162.820, Y  +570.590, Z    +0.000, E1   -55.270, E3 +291173.721}
SPL {X  -162.820, Y  +580.865, Z    +0.000, E1   -55.132, E3 +291189.678}
SPL {X  -162.820, Y  +591.604, Z    +0.000, E1   -55.202, E3 +291204.615}
SPL {X  -162.820, Y  +600.465, Z    +0.000, E1   -55.218, E3 +291217.404}
SPL {X  -162.820, Y  +609.951, Z    +0.000, E1   -55.211, E3 +291231.151}
SPL {X  -162.820, Y  +618.960, Z    +0.000, E1   -55.186, E3 +291244.372}
SPL {X  -162.820, Y  +627.322, Z    +0.000, E1   -55.201, E3 +291256.307}
SPL {X  -162.820, Y  +634.693, Z    +0.000, E1   -55.198, E3 +291267.023}
SPL {X  -162.820, Y  +642.452, Z    +0.000, E1   -55.141, E3 +291278.630}
SPL {X  -162.820, Y  +652.837, Z    +0.000, E1   -55.281, E3 +291292.898}
SPL {X  -162.820, Y  +660.849, Z    +0.000, E1   -55.101, E3 +291305.447}
SPL {X  -162.820, Y  +671.259, Z    +0.000, E1   -55.266, E3 +291319.743}
SPL {X  -162.498, Y  +683.731, Z    +0.000, E1   -55.157, E3 +291338.452}
SPL {X  -161.784, Y  +691.841, Z    +0.000, E1   -55.010, E3 +291350.909}
SPL {X  -161.070, Y  +697.305, Z    +0.000, E1   -54.828, E3 +291359.987}
SPL {X  -159.751, Y  +704.965, Z    +0.000, E1   -54.697, E3 +291371.973}
SPL {X  -158.271, Y  +711.718, Z    +0.000, E1   -54.504, E3 +291382.781}
SPL {X  -157.115, Y  +716.223, Z    +0.000, E1   -54.227, E3 +291390.973}
SPL {X  -155.622, Y  +721.376, Z    +0.000, E1   -53.849, E3 +291400.573}
SPL {X  -153.323, Y  +728.294, Z    +0.000, E1   -53.618, E3 +291412.046}
SPL {X  -150.606, Y  +735.372, Z    +0.000, E1   -53.091, E3 +291425.043}
SPL {X  -148.712, Y  +739.795, Z    +0.000, E1   -52.656, E3 +291433.605}
SPL {X  -146.885, Y  +743.751, Z    +0.000, E1   -52.544, E3 +291439.879}
SPL {X  -144.373, Y  +748.778, Z    +0.000, E1   -52.887, E3 +291445.341}
SPL {X  -137.947, Y  +759.993, Z    +0.000, E1   -55.381, E3 +291448.451}
SPL {X  -123.111, Y  +780.056, Z    +0.000, E1   -48.144, E3 +291547.587}
ENDSPLINE

SPLINE
SPL {X  -146.599, Y  +744.345, Z    +0.000, E1   -36.661, E3 +291632.590}
SPL {X  -157.185, Y  +715.965, Z    +0.000, E1   -25.340, E3 +291635.640}
SPL {X  -159.997, Y  +703.690, Z    +0.000, E1   -19.457, E3 +291636.968}
SPL {X  -161.886, Y  +690.913, Z    +0.000, E1   -12.672, E3 +291641.096}
SPL {X  -162.700, Y  +679.756, Z    +0.000, E1    -6.060, E3 +291640.305}
SPL {X  -162.820, Y  +673.439, Z    +0.000, E1    -1.797, E3 +291640.407}
SPL {X  -162.820, Y  +670.554, Z    +0.000, E1    +0.472, E3 +291639.940}
SPL {X  -162.820, Y  +667.789, Z    +0.000, E1    +3.144, E3 +291639.961}
SPL {X  -162.820, Y  +664.083, Z    +0.000, E1    +7.387, E3 +291639.853}
SPL {X  -162.820, Y  +659.344, Z    +0.000, E1   +13.535, E3 +291639.417}
SPL {X  -162.820, Y  +653.403, Z    +0.000, E1   +21.415, E3 +291639.831}
SPL {X  -162.820, Y  +642.162, Z    +0.000, E1   +35.510, E3 +291639.144}
SPL {X  -162.820, Y  +598.675, Z    +0.000, E1   +56.845, E3 +291656.456}
SPL {X  -162.820, Y  +543.175, Z    +0.000, E1   +54.504, E3 +291732.311}
SPL {X  -162.820, Y  +538.115, Z    +0.000, E1   +53.658, E3 +291745.362}
SPL {X  -162.820, Y  +527.429, Z    +0.000, E1   +53.760, E3 +291761.092}
SPL {X  -162.820, Y  +518.365, Z    +0.000, E1   +53.683, E3 +291775.350}
SPL {X  -162.820, Y  +508.465, Z    +0.000, E1   +53.706, E3 +291790.564}
SPL {X  -162.820, Y  +499.206, Z    +0.000, E1   +53.779, E3 +291804.004}
SPL {X  -162.820, Y  +493.008, Z    +0.000, E1   +53.586, E3 +291814.812}
SPL {X  -162.820, Y  +485.759, Z    +0.000, E1   +53.138, E3 +291828.820}
ENDSPLINE

SPLINE
SPL {X  -162.820, Y  +494.645, Z    +0.000, E1   +48.544, E3 +291841.296}
ENDSPLINE

SPLINE
SPL {X  -162.820, Y  +486.578, Z    +0.000, E1   +49.194, E3 +291852.092}
SPL {X  -162.820, Y  +476.731, Z    +0.000, E1   +50.039, E3 +291864.515}
SPL {X  -162.820, Y  +466.442, Z    +0.000, E1   +50.873, E3 +291877.183}
SPL {X  -162.820, Y  +455.624, Z    +0.000, E1   +51.698, E3 +291890.254}
SPL {X  -162.820, Y  +444.568, Z    +0.000, E1   +52.608, E3 +291902.567}
SPL {X  -162.820, Y  +432.435, Z    +0.000, E1   +53.605, E3 +291915.450}
SPL {X  -162.820, Y  +419.875, Z    +0.000, E1   +54.604, E3 +291928.124}
SPL {X  -162.820, Y  +414.181, Z    +0.000, E1   +54.446, E3 +291937.559}
SPL {X  -162.820, Y  +407.616, Z    +0.000, E1   +54.585, E3 +291946.393}
SPL {X  -162.820, Y  +400.244, Z    +0.000, E1   +54.630, E3 +291957.111}
SPL {X  -162.820, Y  +389.249, Z    +0.000, E1   +54.752, E3 +291972.690}
SPL {X  -162.799, Y  +377.862, Z    +0.000, E1   +54.622, E3 +291990.321}
SPL {X  -162.216, Y  +366.490, Z    +0.000, E1   +54.549, E3 +292007.617}
SPL {X  -160.880, Y  +355.442, Z    +0.000, E1   +54.372, E3 +292025.073}
SPL {X  -159.457, Y  +347.579, Z    +0.000, E1   +54.148, E3 +292037.809}
SPL {X  -158.033, Y  +341.310, Z    +0.000, E1   +53.819, E3 +292049.146}
SPL {X  -155.608, Y  +332.578, Z    +0.000, E1   +53.425, E3 +292064.417}
SPL {X  -152.785, Y  +324.223, Z    +0.000, E1   +52.975, E3 +292079.177}
SPL {X  -150.663, Y  +318.766, Z    +0.000, E1   +52.574, E3 +292089.210}
SPL {X  -148.923, Y  +314.679, Z    +0.000, E1   +52.172, E3 +292097.368}
SPL {X  -146.846, Y  +310.168, Z    +0.000, E1   +51.697, E3 +292106.429}
SPL {X  -140.627, Y  +298.437, Z    +0.000, E1   +54.251, E3 +292110.688}
SPL {X  -122.064, Y  +272.747, Z    +0.000, E1   +48.156, E3 +292216.213}
ENDSPLINE

SPLINE
SPL {X  -148.173, Y  +313.009, Z    +0.000, E1   +35.624, E3 +292299.259}
SPL {X  -158.289, Y  +342.356, Z    +0.000, E1   +23.452, E3 +292302.248}
SPL {X  -161.301, Y  +358.312, Z    +0.000, E1   +15.384, E3 +292304.206}
SPL {X  -162.692, Y  +374.052, Z    +0.000, E1    +6.208, E3 +292304.144}
SPL {X  -162.820, Y  +381.030, Z    +0.000, E1    +1.454, E3 +292304.323}
SPL {X  -162.820, Y  +384.274, Z    +0.000, E1    -1.205, E3 +292304.042}
SPL {X  -162.820, Y  +388.271, Z    +0.000, E1    -5.458, E3 +292304.035}
SPL {X  -162.820, Y  +394.827, Z    +0.000, E1   -13.677, E3 +292303.725}
SPL {X  -162.820, Y  +402.977, Z    +0.000, E1   -24.772, E3 +292304.007}
SPL {X  -162.820, Y  +413.615, Z    +0.000, E1   -37.560, E3 +292303.797}
SPL {X  -162.820, Y  +456.390, Z    +0.000, E1   -57.415, E3 +292320.839}
SPL {X  -162.820, Y  +525.017, Z    +0.000, E1   -58.379, E3 +292391.503}
ENDSPLINE

SPLINE
SPL {X  -162.820, Y  +520.266, Z    +0.000, E1   -55.155, E3 +292405.996}
ENDSPLINE

SPLINE
SPL {X  -162.820, Y  +529.742, Z    +0.000, E1   -55.146, E3 +292419.712}
SPL {X  -162.820, Y  +538.383, Z    +0.000, E1   -55.306, E3 +292431.164}
SPL {X  -162.820, Y  +544.790, Z    +0.000, E1   -55.066, E3 +292441.964}
SPL {X  -162.820, Y  +555.105, Z    +0.000, E1   -55.222, E3 +292456.085}
SPL {X  -162.820, Y  +563.355, Z    +0.000, E1   -55.172, E3 +292468.151}
SPL {X  -162.820, Y  +570.590, Z    +0.000, E1   -55.270, E3 +292478.069}
SPL {X  -162.820, Y  +580.865, Z    +0.000, E1   -55.132, E3 +292494.026}
SPL {X  -162.820, Y  +591.604, Z    +0.000, E1   -55.202, E3 +292508.963}
SPL {X  -162.820, Y  +600.465, Z    +0.000, E1   -55.218, E3 +292521.752}
SPL {X  -162.820, Y  +609.951, Z    +0.000, E1   -55.211, E3 +292535.499}
SPL {X  -162.820, Y  +617.278, Z    +0.000, E1   -55.256, E3 +292545.723}
SPL {X  -162.820, Y  +625.209, Z    +0.000, E1   -55.167, E3 +292557.915}
SPL {X  -162.820, Y  +634.693, Z    +0.000, E1   -55.198, E3 +292571.371}
SPL {X  -162.820, Y  +642.452, Z    +0.000, E1   -55.141, E3 +292582.978}
SPL {X  -162.820, Y  +652.837, Z    +0.000, E1   -55.281, E3 +292597.246}
SPL {X  -162.820, Y  +660.849, Z    +0.000, E1   -55.101, E3 +292609.795}
SPL {X  -162.820, Y  +671.259, Z    +0.000, E1   -55.266, E3 +292624.090}
SPL {X  -162.498, Y  +683.731, Z    +0.000, E1   -55.157, E3 +292642.800}
SPL {X  -161.784, Y  +691.841, Z    +0.000, E1   -55.010, E3 +292655.257}
SPL {X  -161.070, Y  +697.305, Z    +0.000, E1   -54.828, E3 +292664.335}
SPL {X  -159.751, Y  +704.965, Z    +0.000, E1   -54.697, E3 +292676.321}
SPL {X  -158.271, Y  +711.718, Z    +0.000, E1   -54.504, E3 +292687.129}
SPL {X  -157.115, Y  +716.223, Z    +0.000, E1   -54.227, E3 +292695.321}
SPL {X  -155.622, Y  +721.376, Z    +0.000, E1   -53.849, E3 +292704.921}
SPL {X  -153.323, Y  +728.294, Z    +0.000, E1   -53.618, E3 +292716.394}
SPL {X  -150.606, Y  +735.372, Z    +0.000, E1   -53.091, E3 +292729.391}
SPL {X  -148.712, Y  +739.795, Z    +0.000, E1   -52.656, E3 +292737.953}
SPL {X  -146.885, Y  +743.751, Z    +0.000, E1   -52.544, E3 +292744.227}
SPL {X  -144.373, Y  +748.778, Z    +0.000, E1   -52.887, E3 +292749.689}
SPL {X  -137.947, Y  +759.993, Z    +0.000, E1   -55.381, E3 +292752.799}
SPL {X  -123.111, Y  +780.056, Z    +0.000, E1   -48.144, E3 +292851.935}
ENDSPLINE

SPLINE
SPL {X  -146.599, Y  +744.345, Z    +0.000, E1   -36.661, E3 +292936.938}
SPL {X  -158.886, Y  +709.076, Z    +0.000, E1   -22.176, E3 +292940.810}
SPL {X  -161.886, Y  +690.913, Z    +0.000, E1   -12.672, E3 +292945.444}
SPL {X  -162.573, Y  +682.458, Z    +0.000, E1    -7.683, E3 +292944.945}
SPL {X  -162.817, Y  +674.426, Z    +0.000, E1    -2.573, E3 +292944.663}
SPL {X  -162.820, Y  +670.554, Z    +0.000, E1    +0.472, E3 +292944.288}
SPL {X  -162.820, Y  +667.789, Z    +0.000, E1    +3.144, E3 +292944.309}
SPL {X  -162.820, Y  +664.083, Z    +0.000, E1    +7.387, E3 +292944.201}
SPL {X  -162.820, Y  +659.344, Z    +0.000, E1   +13.535, E3 +292943.765}
SPL {X  -162.820, Y  +653.403, Z    +0.000, E1   +21.415, E3 +292944.179}
SPL {X  -162.820, Y  +644.970, Z    +0.000, E1   +32.346, E3 +292943.596}
SPL {X  -162.820, Y  +637.013, Z    +0.000, E1   +41.185, E3 +292943.301}
SPL {X  -162.820, Y  +603.840, Z    +0.000, E1   +55.833, E3 +292957.917}
SPL {X  -162.820, Y  +590.612, Z    +0.000, E1   +58.217, E3 +292965.301}
SPL {X  -162.820, Y  +543.175, Z    +0.000, E1   +54.504, E3 +293036.659}
SPL {X  -162.820, Y  +538.115, Z    +0.000, E1   +53.658, E3 +293049.710}
SPL {X  -162.820, Y  +527.429, Z    +0.000, E1   +53.760, E3 +293065.440}
SPL {X  -162.820, Y  +518.365, Z    +0.000, E1   +53.683, E3 +293079.698}
SPL {X  -162.820, Y  +510.654, Z    +0.000, E1   +53.658, E3 +293091.697}
SPL {X  -162.820, Y  +501.304, Z    +0.000, E1   +53.758, E3 +293105.385}
SPL {X  -162.820, Y  +493.008, Z    +0.000, E1   +53.586, E3 +293119.160}
SPL {X  -162.820, Y  +485.759, Z    +0.000, E1   +53.138, E3 +293133.168}
ENDSPLINE

SPLINE
SPL {X  -162.820, Y  +494.645, Z    +0.000, E1   +48.544, E3 +293145.644}
ENDSPLINE

SPLINE
SPL {X  -162.820, Y  +486.578, Z    +0.000, E1   +49.194, E3 +293156.440}
SPL {X  -162.820, Y  +476.731, Z    +0.000, E1   +50.039, E3 +293168.863}
SPL {X  -162.820, Y  +466.442, Z    +0.000, E1   +50.873, E3 +293181.531}
SPL {X  -162.820, Y  +455.624, Z    +0.000, E1   +51.698, E3 +293194.602}
SPL {X  -162.820, Y  +444.568, Z    +0.000, E1   +52.608, E3 +293206.915}
SPL {X  -162.820, Y  +432.435, Z    +0.000, E1   +53.605, E3 +293219.798}
SPL {X  -162.820, Y  +419.900, Z    +0.000, E1   +54.598, E3 +293232.473}
SPL {X  -162.820, Y  +411.092, Z    +0.000, E1   +54.552, E3 +293245.993}
SPL {X  -162.820, Y  +400.244, Z    +0.000, E1   +54.630, E3 +293261.459}
SPL {X  -162.820, Y  +392.496, Z    +0.000, E1   +54.734, E3 +293272.160}
SPL {X  -162.820, Y  +387.085, Z    +0.000, E1   +54.699, E3 +293280.387}
SPL {X  -162.820, Y  +380.650, Z    +0.000, E1   +54.601, E3 +293290.483}
SPL {X  -162.727, Y  +374.992, Z    +0.000, E1   +54.549, E3 +293299.165}
SPL {X  -162.216, Y  +366.490, Z    +0.000, E1   +54.549, E3 +293311.964}
SPL {X  -160.880, Y  +355.442, Z    +0.000, E1   +54.372, E3 +293329.421}
SPL {X  -159.457, Y  +347.579, Z    +0.000, E1   +54.148, E3 +293342.157}
SPL {X  -158.033, Y  +341.310, Z    +0.000, E1   +53.819, E3 +293353.494}
SPL {X  -155.608, Y  +332.578, Z    +0.000, E1   +53.425, E3 +293368.765}
SPL {X  -153.385, Y  +325.878, Z    +0.000, E1   +53.068, E3 +293380.433}
SPL {X  -151.310, Y  +320.369, Z    +0.000, E1   +52.706, E3 +293390.631}
SPL {X  -148.923, Y  +314.679, Z    +0.000, E1   +52.172, E3 +293401.716}
SPL {X  -146.846, Y  +310.168, Z    +0.000, E1   +51.697, E3 +293410.777}
SPL {X  -140.627, Y  +298.437, Z    +0.000, E1   +54.251, E3 +293415.036}
SPL {X  -122.064, Y  +272.747, Z    +0.000, E1   +48.156, E3 +293520.561}
ENDSPLINE

SPLINE
SPL {X  -148.173, Y  +313.009, Z    +0.000, E1   +35.624, E3 +293603.607}
SPL {X  -158.289, Y  +342.356, Z    +0.000, E1   +23.452, E3 +293606.596}
SPL {X  -161.301, Y  +358.312, Z    +0.000, E1   +15.384, E3 +293608.554}
SPL {X  -162.692, Y  +374.052, Z    +0.000, E1    +6.208, E3 +293608.492}
SPL {X  -162.820, Y  +381.030, Z    +0.000, E1    +1.454, E3 +293608.671}
SPL {X  -162.820, Y  +384.274, Z    +0.000, E1    -1.205, E3 +293608.390}
SPL {X  -162.820, Y  +388.271, Z    +0.000, E1    -5.458, E3 +293608.382}
SPL {X  -162.820, Y  +394.827, Z    +0.000, E1   -13.677, E3 +293608.073}
SPL {X  -162.820, Y  +402.977, Z    +0.000, E1   -24.772, E3 +293608.354}
SPL {X  -162.820, Y  +413.615, Z    +0.000, E1   -37.560, E3 +293608.145}
SPL {X  -162.820, Y  +456.390, Z    +0.000, E1   -57.415, E3 +293625.186}
SPL {X  -162.820, Y  +525.017, Z    +0.000, E1   -58.379, E3 +293695.851}
ENDSPLINE

SPLINE
SPL {X  -162.820, Y  +515.796, Z    +0.000, E1   -54.952, E3 +293704.958}
ENDSPLINE

SPLINE
SPL {X  -162.820, Y  +522.537, Z    +0.000, E1   -55.218, E3 +293713.133}
SPL {X  -162.820, Y  +529.742, Z    +0.000, E1   -55.146, E3 +293724.060}
SPL {X  -162.820, Y  +538.383, Z    +0.000, E1   -55.306, E3 +293735.512}
SPL {X  -162.820, Y  +544.790, Z    +0.000, E1   -55.066, E3 +293746.312}
SPL {X  -162.820, Y  +552.981, Z    +0.000, E1   -55.286, E3 +293756.775}
SPL {X  -162.820, Y  +560.767, Z    +0.000, E1   -55.137, E3 +293769.083}
SPL {X  -162.820, Y  +570.590, Z    +0.000, E1   -55.270, E3 +293782.417}
SPL {X  -162.820, Y  +577.946, Z    +0.000, E1   -55.110, E3 +293794.055}
SPL {X  -162.820, Y  +583.981, Z    +0.000, E1   -55.057, E3 +293803.137}
SPL {X  -162.820, Y  +591.604, Z    +0.000, E1   -55.202, E3 +293813.311}
SPL {X  -162.820, Y  +600.465, Z    +0.000, E1   -55.218, E3 +293826.099}
SPL {X  -162.820, Y  +609.951, Z    +0.000, E1   -55.211, E3 +293839.847}
SPL {X  -162.820, Y  +617.278, Z    +0.000, E1   -55.256, E3 +293850.071}
SPL {X  -162.820, Y  +625.209, Z    +0.000, E1   -55.167, E3 +293862.263}
SPL {X  -162.820, Y  +634.693, Z    +0.000, E1   -55.198, E3 +293875.719}
SPL {X  -162.820, Y  +642.452, Z    +0.000, E1   -55.141, E3 +293887.326}
SPL {X  -162.820, Y  +652.837, Z    +0.000, E1   -55.281, E3 +293901.594}
SPL {X  -162.820, Y  +660.849, Z    +0.000, E1   -55.101, E3 +293914.143}
SPL {X  -162.820, Y  +668.534, Z    +0.000, E1   -55.182, E3 +293924.856}
SPL {X  -162.763, Y  +677.803, Z    +0.000, E1   -55.175, E3 +293938.362}
SPL {X  -162.314, Y  +686.325, Z    +0.000, E1   -55.173, E3 +293950.642}
SPL {X  -161.784, Y  +691.841, Z    +0.000, E1   -55.010, E3 +293959.604}
SPL {X  -161.070, Y  +697.305, Z    +0.000, E1   -54.828, E3 +293968.682}
SPL {X  -159.751, Y  +704.965, Z    +0.000, E1   -54.697, E3 +293980.668}
SPL {X  -158.271, Y  +711.718, Z    +0.000, E1   -54.504, E3 +293991.477}
SPL {X  -157.115, Y  +716.223, Z    +0.000, E1   -54.227, E3 +293999.669}
SPL {X  -154.825, Y  +723.894, Z    +0.000, E1   -53.830, E3 +294013.209}
SPL {X  -152.160, Y  +731.445, Z    +0.000, E1   -53.336, E3 +294026.751}
SPL {X  -149.361, Y  +738.321, Z    +0.000, E1   -52.873, E3 +294039.214}
SPL {X  -146.885, Y  +743.751, Z    +0.000, E1   -52.544, E3 +294048.575}
SPL {X  -144.373, Y  +748.778, Z    +0.000, E1   -52.887, E3 +294054.037}
SPL {X  -137.947, Y  +759.993, Z    +0.000, E1   -55.381, E3 +294057.147}
SPL {X  -123.111, Y  +780.056, Z    +0.000, E1   -48.144, E3 +294156.282}
ENDSPLINE

SPLINE
SPL {X  -146.599, Y  +744.345, Z    +0.000, E1   -36.661, E3 +294241.286}
SPL {X  -157.185, Y  +715.965, Z    +0.000, E1   -25.340, E3 +294244.336}
SPL {X  -159.997, Y  +703.690, Z    +0.000, E1   -19.457, E3 +294245.664}
SPL {X  -161.886, Y  +690.913, Z    +0.000, E1   -12.672, E3 +294249.792}
SPL {X  -162.700, Y  +679.756, Z    +0.000, E1    -6.060, E3 +294249.001}
SPL {X  -162.820, Y  +673.439, Z    +0.000, E1    -1.797, E3 +294249.103}
SPL {X  -162.820, Y  +670.554, Z    +0.000, E1    +0.472, E3 +294248.635}
SPL {X  -162.820, Y  +667.789, Z    +0.000, E1    +3.144, E3 +294248.657}
SPL {X  -162.820, Y  +664.083, Z    +0.000, E1    +7.387, E3 +294248.549}
SPL {X  -162.820, Y  +659.344, Z    +0.000, E1   +13.535, E3 +294248.112}
SPL {X  -162.820, Y  +653.403, Z    +0.000, E1   +21.415, E3 +294248.527}
SPL {X  -162.820, Y  +642.162, Z    +0.000, E1   +35.510, E3 +294247.839}
SPL {X  -162.820, Y  +598.675, Z    +0.000, E1   +56.845, E3 +294265.152}
SPL {X  -162.820, Y  +543.175, Z    +0.000, E1   +54.504, E3 +294341.006}
SPL {X  -162.820, Y  +538.115, Z    +0.000, E1   +53.658, E3 +294354.058}
SPL {X  -162.820, Y  +530.332, Z    +0.000, E1   +53.757, E3 +294365.201}
SPL {X  -162.820, Y  +525.300, Z    +0.000, E1   +53.701, E3 +294373.252}
SPL {X  -162.820, Y  +518.365, Z    +0.000, E1   +53.683, E3 +294384.045}
SPL {X  -162.820, Y  +510.654, Z    +0.000, E1   +53.658, E3 +294396.044}
SPL {X  -162.820, Y  +501.304, Z    +0.000, E1   +53.758, E3 +294409.733}
SPL {X  -162.820, Y  +493.008, Z    +0.000, E1   +53.586, E3 +294423.508}
SPL {X  -162.820, Y  +484.615, Z    +0.000, E1   +53.726, E3 +294435.439}
ENDSPLINE

SPLINE
SPL {X  -162.820, Y  +492.996, Z    +0.000, E1   +49.430, E3 +294447.985}
ENDSPLINE

SPLINE
SPL {X  -162.820, Y  +486.578, Z    +0.000, E1   +49.194, E3 +294460.788}
SPL {X  -162.820, Y  +476.731, Z    +0.000, E1   +50.039, E3 +294473.211}
SPL {X  -162.820, Y  +466.442, Z    +0.000, E1   +50.873, E3 +294485.879}
SPL {X  -162.820, Y  +455.624, Z    +0.000, E1   +51.698, E3 +294498.950}
SPL {X  -162.820, Y  +444.568, Z    +0.000, E1   +52.608, E3 +294511.263}
SPL {X  -162.820, Y  +432.435, Z    +0.000, E1   +53.605, E3 +294524.146}
SPL {X  -162.820, Y  +419.875, Z    +0.000, E1   +54.604, E3 +294536.820}
SPL {X  -162.820, Y  +414.181, Z    +0.000, E1   +54.446, E3 +294546.255}
SPL {X  -162.820, Y  +407.616, Z    +0.000, E1   +54.585, E3 +294555.089}
SPL {X  -162.820, Y  +400.244, Z    +0.000, E1   +54.630, E3 +294565.807}
SPL {X  -162.820, Y  +389.249, Z    +0.000, E1   +54.752, E3 +294581.386}
SPL {X  -162.820, Y  +380.650, Z    +0.000, E1   +54.601, E3 +294594.831}
SPL {X  -162.727, Y  +374.992, Z    +0.000, E1   +54.549, E3 +294603.513}
SPL {X  -162.373, Y  +368.447, Z    +0.000, E1   +54.597, E3 +294612.945}
SPL {X  -161.939, Y  +363.587, Z    +0.000, E1   +54.355, E3 +294621.558}
SPL {X  -160.880, Y  +355.442, Z    +0.000, E1   +54.372, E3 +294633.769}
SPL {X  -159.457, Y  +347.579, Z    +0.000, E1   +54.148, E3 +294646.505}
SPL {X  -158.033, Y  +341.310, Z    +0.000, E1   +53.819, E3 +294657.842}
SPL {X  -156.195, Y  +334.528, Z    +0.000, E1   +53.534, E3 +294669.407}
SPL {X  -154.120, Y  +327.988, Z    +0.000, E1   +53.171, E3 +294681.264}
SPL {X  -151.310, Y  +320.369, Z    +0.000, E1   +52.706, E3 +294694.979}
SPL {X  -148.923, Y  +314.679, Z    +0.000, E1   +52.172, E3 +294706.064}
SPL {X  -146.846, Y  +310.168, Z    +0.000, E1   +51.697, E3 +294715.125}
SPL {X  -140.627, Y  +298.437, Z    +0.000, E1   +54.251, E3 +294719.384}
SPL {X  -122.064, Y  +272.747, Z    +0.000, E1   +48.156, E3 +294824.909}
ENDSPLINE

